    movel([0.115711, -1.231258, -2.664725, -0.816406, 1.570796, 1.686507],accel_mss,speed_ms,0,blend_radius_m)
    movel([0.117256, -1.231856, -2.664420, -0.816113, 1.570796, 1.688052],accel_mss,speed_ms,0,blend_radius_m)
    movel([0.117989, -1.233200, -2.663733, -0.815456, 1.570796, 1.688785],accel_mss,speed_ms,0,blend_radius_m)
    movel([0.117965, -1.234308, -2.663164, -0.814916, 1.570796, 1.688761],accel_mss,speed_ms,0,blend_radius_m)
    movel([0.117577, -1.235608, -2.662496, -0.814285, 1.570796, 1.688373],accel_mss,speed_ms,0,blend_radius_m)
    movel([0.116887, -1.236930, -2.661814, -0.813645, 1.570796, 1.687683],accel_mss,speed_ms,0,blend_radius_m)
    movel([0.115976, -1.238105, -2.661207, -0.813078, 1.570796, 1.686772],accel_mss,speed_ms,0,blend_radius_m)
    movel([0.115156, -1.238911, -2.660789, -0.812690, 1.570796, 1.685952],accel_mss,speed_ms,0,blend_radius_m)
    movel([0.114390, -1.239502, -2.660482, -0.812406, 1.570796, 1.685186],accel_mss,speed_ms,0,blend_radius_m)
    movel([0.113558, -1.239966, -2.660241, -0.812183, 1.570796, 1.684355],accel_mss,speed_ms,0,blend_radius_m)
    movel([0.112538, -1.240377, -2.660026, -0.811985, 1.570796, 1.683335],accel_mss,speed_ms,0,blend_radius_m)
    movel([0.111513, -1.240676, -2.659871, -0.811842, 1.570796, 1.682309],accel_mss,speed_ms,0,blend_radius_m)
    movel([0.110720, -1.240770, -2.659822, -0.811797, 1.570796, 1.681516],accel_mss,speed_ms,0,blend_radius_m)
    movel([0.110024, -1.240667, -2.659876, -0.811847, 1.570796, 1.680820],accel_mss,speed_ms,0,blend_radius_m)
    movel([0.109302, -1.240359, -2.660036, -0.811994, 1.570796, 1.680098],accel_mss,speed_ms,0,blend_radius_m)
    movel([0.108717, -1.239916, -2.660266, -0.812206, 1.570796, 1.679513],accel_mss,speed_ms,0,blend_radius_m)
    movel([0.108365, -1.239370, -2.660550, -0.812468, 1.570796, 1.679162],accel_mss,speed_ms,0,blend_radius_m)
    movel([0.108218, -1.238654, -2.660922, -0.812813, 1.570796, 1.679014],accel_mss,speed_ms,0,blend_radius_m)
    movel([0.108256, -1.237694, -2.661419, -0.813276, 1.570796, 1.679053],accel_mss,speed_ms,0,blend_radius_m)
    movel([0.108349, -1.237041, -2.661757, -0.813591, 1.570796, 1.679145],accel_mss,speed_ms,0,blend_radius_m)
    movel([0.108457, -1.236591, -2.661989, -0.813809, 1.570796, 1.679253],accel_mss,speed_ms,0,blend_radius_m)
    movel([0.108621, -1.236171, -2.662206, -0.814012, 1.570796, 1.679418],accel_mss,speed_ms,0,blend_radius_m)
    movel([0.108896, -1.235638, -2.662480, -0.814270, 1.570796, 1.679692],accel_mss,speed_ms,0,blend_radius_m)
    movel([0.109412, -1.234833, -2.662895, -0.814661, 1.570796, 1.680209],accel_mss,speed_ms,0,blend_radius_m)
    speed_ms = 0.003
    movel([0.109412, -1.220507, -2.655895, -0.835988, 1.570796, 1.680209],accel_mss,speed_ms,0,blend_radius_m)
    speed_ms = 1.000
    movel([0.109412, -1.193393, -2.641522, -0.877474, 1.570796, 1.680209],accel_mss,speed_ms,0,blend_radius_m)
    movel([0.123315, -1.189342, -2.643484, -0.879564, 1.570796, 1.694112],accel_mss,speed_ms,0,blend_radius_m)
    movel([0.123315, -1.216492, -2.657910, -0.837988, 1.570796, 1.694112],accel_mss,speed_ms,0,blend_radius_m)
    speed_ms = 0.003
    movel([0.123315, -1.227206, -2.663192, -0.821991, 1.570796, 1.694112],accel_mss,speed_ms,0,blend_radius_m)
    speed_ms = 0.007
    movel([0.123570, -1.225425, -2.664093, -0.822871, 1.570796, 1.694367],accel_mss,speed_ms,0,blend_radius_m)
    movel([0.123913, -1.223185, -2.665221, -0.823983, 1.570796, 1.694710],accel_mss,speed_ms,0,blend_radius_m)
    movel([0.124125, -1.222339, -2.665645, -0.824405, 1.570796, 1.694921],accel_mss,speed_ms,0,blend_radius_m)
    movel([0.124611, -1.222347, -2.665641, -0.824401, 1.570796, 1.695407],accel_mss,speed_ms,0,blend_radius_m)
    movel([0.124874, -1.223146, -2.665240, -0.824003, 1.570796, 1.695670],accel_mss,speed_ms,0,blend_radius_m)
    movel([0.124930, -1.224185, -2.664718, -0.823486, 1.570796, 1.695726],accel_mss,speed_ms,0,blend_radius_m)
    movel([0.124787, -1.225358, -2.664126, -0.822904, 1.570796, 1.695583],accel_mss,speed_ms,0,blend_radius_m)
    movel([0.124446, -1.226559, -2.663520, -0.822311, 1.570796, 1.695243],accel_mss,speed_ms,0,blend_radius_m)
    movel([0.124141, -1.227337, -2.663125, -0.821927, 1.570796, 1.694937],accel_mss,speed_ms,0,blend_radius_m)
    movel([0.123839, -1.227943, -2.662818, -0.821628, 1.570796, 1.694636],accel_mss,speed_ms,0,blend_radius_m)
    movel([0.123561, -1.228363, -2.662604, -0.821421, 1.570796, 1.694357],accel_mss,speed_ms,0,blend_radius_m)
    movel([0.123214, -1.228488, -2.662541, -0.821360, 1.570796, 1.694010],accel_mss,speed_ms,0,blend_radius_m)
    movel([0.123227, -1.228032, -2.662773, -0.821584, 1.570796, 1.694023],accel_mss,speed_ms,0,blend_radius_m)
    movel([0.123315, -1.227206, -2.663192, -0.821991, 1.570796, 1.694112],accel_mss,speed_ms,0,blend_radius_m)
    speed_ms = 0.003
    movel([0.123315, -1.230843, -2.664937, -0.816609, 1.570796, 1.694112],accel_mss,speed_ms,0,blend_radius_m)
    speed_ms = 0.007
    movel([0.123570, -1.229065, -2.665841, -0.817483, 1.570796, 1.694367],accel_mss,speed_ms,0,blend_radius_m)
    movel([0.123913, -1.226829, -2.666972, -0.818588, 1.570796, 1.694710],accel_mss,speed_ms,0,blend_radius_m)
    movel([0.124125, -1.225985, -2.667398, -0.819006, 1.570796, 1.694921],accel_mss,speed_ms,0,blend_radius_m)
    movel([0.124611, -1.225992, -2.667394, -0.819002, 1.570796, 1.695407],accel_mss,speed_ms,0,blend_radius_m)
    movel([0.124874, -1.226790, -2.666992, -0.818607, 1.570796, 1.695670],accel_mss,speed_ms,0,blend_radius_m)
    movel([0.124930, -1.227827, -2.666468, -0.818094, 1.570796, 1.695726],accel_mss,speed_ms,0,blend_radius_m)
    movel([0.124787, -1.228999, -2.665874, -0.817516, 1.570796, 1.695583],accel_mss,speed_ms,0,blend_radius_m)
    movel([0.124446, -1.230197, -2.665265, -0.816926, 1.570796, 1.695243],accel_mss,speed_ms,0,blend_radius_m)
    movel([0.124141, -1.230974, -2.664870, -0.816545, 1.570796, 1.694937],accel_mss,speed_ms,0,blend_radius_m)
    movel([0.123839, -1.231579, -2.664561, -0.816248, 1.570796, 1.694636],accel_mss,speed_ms,0,blend_radius_m)
    movel([0.123561, -1.231999, -2.664347, -0.816043, 1.570796, 1.694357],accel_mss,speed_ms,0,blend_radius_m)
    movel([0.123214, -1.232124, -2.664283, -0.815982, 1.570796, 1.694010],accel_mss,speed_ms,0,blend_radius_m)
    movel([0.123227, -1.231668, -2.664516, -0.816205, 1.570796, 1.694023],accel_mss,speed_ms,0,blend_radius_m)
    movel([0.123315, -1.230843, -2.664937, -0.816609, 1.570796, 1.694112],accel_mss,speed_ms,0,blend_radius_m)
    speed_ms = 0.003
    movel([0.123315, -1.216492, -2.657910, -0.837988, 1.570796, 1.694112],accel_mss,speed_ms,0,blend_radius_m)
    speed_ms = 1.000
    movel([0.123315, -1.189342, -2.643484, -0.879564, 1.570796, 1.694112],accel_mss,speed_ms,0,blend_radius_m)
    movel([0.125124, -1.188800, -2.643744, -0.879845, 1.570796, 1.695920],accel_mss,speed_ms,0,blend_radius_m)
    movel([0.125124, -1.215955, -2.658178, -0.838257, 1.570796, 1.695920],accel_mss,speed_ms,0,blend_radius_m)
    speed_ms = 0.003
    movel([0.125124, -1.226671, -2.663463, -0.822255, 1.570796, 1.695920],accel_mss,speed_ms,0,blend_radius_m)
    speed_ms = 0.007
    movel([0.125227, -1.226209, -2.663697, -0.822484, 1.570796, 1.696023],accel_mss,speed_ms,0,blend_radius_m)
    movel([0.125307, -1.225911, -2.663847, -0.822631, 1.570796, 1.696104],accel_mss,speed_ms,0,blend_radius_m)
    movel([0.125412, -1.225400, -2.664105, -0.822884, 1.570796, 1.696208],accel_mss,speed_ms,0,blend_radius_m)
    movel([0.125518, -1.224812, -2.664402, -0.823175, 1.570796, 1.696314],accel_mss,speed_ms,0,blend_radius_m)
    movel([0.125611, -1.224215, -2.664703, -0.823471, 1.570796, 1.696408],accel_mss,speed_ms,0,blend_radius_m)
    movel([0.125825, -1.222759, -2.665435, -0.824196, 1.570796, 1.696622],accel_mss,speed_ms,0,blend_radius_m)
    movel([0.126387, -1.222525, -2.665552, -0.824312, 1.570796, 1.697183],accel_mss,speed_ms,0,blend_radius_m)
    movel([0.127048, -1.222423, -2.665603, -0.824363, 1.570796, 1.697844],accel_mss,speed_ms,0,blend_radius_m)
    movel([0.127393, -1.222737, -2.665446, -0.824207, 1.570796, 1.698189],accel_mss,speed_ms,0,blend_radius_m)
    movel([0.127359, -1.223478, -2.665074, -0.823837, 1.570796, 1.698155],accel_mss,speed_ms,0,blend_radius_m)
    movel([0.126927, -1.224592, -2.664513, -0.823284, 1.570796, 1.697723],accel_mss,speed_ms,0,blend_radius_m)
    movel([0.126733, -1.224966, -2.664324, -0.823099, 1.570796, 1.697529],accel_mss,speed_ms,0,blend_radius_m)
    movel([0.126474, -1.225394, -2.664108, -0.822887, 1.570796, 1.697270],accel_mss,speed_ms,0,blend_radius_m)
    movel([0.126203, -1.225807, -2.663900, -0.822682, 1.570796, 1.696999],accel_mss,speed_ms,0,blend_radius_m)
    movel([0.125955, -1.226134, -2.663735, -0.822521, 1.570796, 1.696752],accel_mss,speed_ms,0,blend_radius_m)
    movel([0.125504, -1.226643, -2.663477, -0.822269, 1.570796, 1.696300],accel_mss,speed_ms,0,blend_radius_m)
    movel([0.125124, -1.226671, -2.663463, -0.822255, 1.570796, 1.695920],accel_mss,speed_ms,0,blend_radius_m)
    speed_ms = 0.003
    movel([0.125124, -1.230310, -2.665208, -0.816871, 1.570796, 1.695920],accel_mss,speed_ms,0,blend_radius_m)
    speed_ms = 0.007
    movel([0.125227, -1.229848, -2.665443, -0.817098, 1.570796, 1.696023],accel_mss,speed_ms,0,blend_radius_m)
    movel([0.125307, -1.229550, -2.665594, -0.817244, 1.570796, 1.696104],accel_mss,speed_ms,0,blend_radius_m)
    movel([0.125412, -1.229040, -2.665853, -0.817495, 1.570796, 1.696208],accel_mss,speed_ms,0,blend_radius_m)
    movel([0.125518, -1.228453, -2.666151, -0.817785, 1.570796, 1.696314],accel_mss,speed_ms,0,blend_radius_m)
    movel([0.125611, -1.227857, -2.666453, -0.818079, 1.570796, 1.696408],accel_mss,speed_ms,0,blend_radius_m)
    movel([0.125825, -1.226403, -2.667187, -0.818798, 1.570796, 1.696622],accel_mss,speed_ms,0,blend_radius_m)
    movel([0.126387, -1.226170, -2.667305, -0.818914, 1.570796, 1.697183],accel_mss,speed_ms,0,blend_radius_m)
    movel([0.127048, -1.226069, -2.667356, -0.818964, 1.570796, 1.697844],accel_mss,speed_ms,0,blend_radius_m)
    movel([0.127393, -1.226381, -2.667198, -0.818809, 1.570796, 1.698189],accel_mss,speed_ms,0,blend_radius_m)
    movel([0.127359, -1.227122, -2.666825, -0.818443, 1.570796, 1.698155],accel_mss,speed_ms,0,blend_radius_m)
    movel([0.126927, -1.228234, -2.666262, -0.817893, 1.570796, 1.697723],accel_mss,speed_ms,0,blend_radius_m)
    movel([0.126733, -1.228607, -2.666073, -0.817709, 1.570796, 1.697529],accel_mss,speed_ms,0,blend_radius_m)
    movel([0.126474, -1.229034, -2.665856, -0.817498, 1.570796, 1.697270],accel_mss,speed_ms,0,blend_radius_m)
    movel([0.126203, -1.229447, -2.665647, -0.817295, 1.570796, 1.696999],accel_mss,speed_ms,0,blend_radius_m)
    movel([0.125955, -1.229773, -2.665481, -0.817135, 1.570796, 1.696752],accel_mss,speed_ms,0,blend_radius_m)
    movel([0.125504, -1.230281, -2.665223, -0.816885, 1.570796, 1.696300],accel_mss,speed_ms,0,blend_radius_m)
    movel([0.125124, -1.230310, -2.665208, -0.816871, 1.570796, 1.695920],accel_mss,speed_ms,0,blend_radius_m)
    speed_ms = 0.003
    movel([0.125124, -1.215955, -2.658178, -0.838257, 1.570796, 1.695920],accel_mss,speed_ms,0,blend_radius_m)
    speed_ms = 1.000
    movel([0.125124, -1.188800, -2.643744, -0.879845, 1.570796, 1.695920],accel_mss,speed_ms,0,blend_radius_m)
    movel([0.132047, -1.189022, -2.643637, -0.879729, 1.570796, 1.702844],accel_mss,speed_ms,0,blend_radius_m)
    movel([0.132047, -1.216175, -2.658068, -0.838146, 1.570796, 1.702844],accel_mss,speed_ms,0,blend_radius_m)
    speed_ms = 0.003
    movel([0.132047, -1.226891, -2.663351, -0.822147, 1.570796, 1.702844],accel_mss,speed_ms,0,blend_radius_m)
    speed_ms = 0.007
    movel([0.132638, -1.225634, -2.663987, -0.822768, 1.570796, 1.703435],accel_mss,speed_ms,0,blend_radius_m)
    movel([0.133199, -1.224453, -2.664583, -0.823353, 1.570796, 1.703995],accel_mss,speed_ms,0,blend_radius_m)
    movel([0.133706, -1.223415, -2.665105, -0.823869, 1.570796, 1.704502],accel_mss,speed_ms,0,blend_radius_m)
    movel([0.134145, -1.222533, -2.665548, -0.824308, 1.570796, 1.704942],accel_mss,speed_ms,0,blend_radius_m)
    movel([0.134644, -1.222071, -2.665779, -0.824538, 1.570796, 1.705440],accel_mss,speed_ms,0,blend_radius_m)
    movel([0.137265, -1.221154, -2.666238, -0.824996, 1.570796, 1.708061],accel_mss,speed_ms,0,blend_radius_m)
    movel([0.139899, -1.220261, -2.666685, -0.825444, 1.570796, 1.710696],accel_mss,speed_ms,0,blend_radius_m)
    movel([0.140179, -1.220315, -2.666657, -0.825416, 1.570796, 1.710976],accel_mss,speed_ms,0,blend_radius_m)
    movel([0.139664, -1.221322, -2.666155, -0.824913, 1.570796, 1.710461],accel_mss,speed_ms,0,blend_radius_m)
    movel([0.139060, -1.222362, -2.665634, -0.824393, 1.570796, 1.709856],accel_mss,speed_ms,0,blend_radius_m)
    movel([0.138330, -1.223574, -2.665025, -0.823790, 1.570796, 1.709127],accel_mss,speed_ms,0,blend_radius_m)
    movel([0.137599, -1.224793, -2.664411, -0.823184, 1.570796, 1.708395],accel_mss,speed_ms,0,blend_radius_m)
    movel([0.136986, -1.225855, -2.663875, -0.822658, 1.570796, 1.707782],accel_mss,speed_ms,0,blend_radius_m)
    movel([0.136486, -1.226755, -2.663420, -0.822214, 1.570796, 1.707282],accel_mss,speed_ms,0,blend_radius_m)
    movel([0.136518, -1.227033, -2.663280, -0.822077, 1.570796, 1.707315],accel_mss,speed_ms,0,blend_radius_m)
    movel([0.137154, -1.226936, -2.663329, -0.822124, 1.570796, 1.707950],accel_mss,speed_ms,0,blend_radius_m)
    movel([0.138087, -1.226651, -2.663473, -0.822265, 1.570796, 1.708883],accel_mss,speed_ms,0,blend_radius_m)
    movel([0.139264, -1.226294, -2.663654, -0.822441, 1.570796, 1.710060],accel_mss,speed_ms,0,blend_radius_m)
    movel([0.139772, -1.226178, -2.663712, -0.822499, 1.570796, 1.710568],accel_mss,speed_ms,0,blend_radius_m)
    movel([0.140019, -1.226346, -2.663627, -0.822416, 1.570796, 1.710815],accel_mss,speed_ms,0,blend_radius_m)
    movel([0.138614, -1.228269, -2.662652, -0.821468, 1.570796, 1.709410],accel_mss,speed_ms,0,blend_radius_m)
    movel([0.137118, -1.230263, -2.661637, -0.820489, 1.570796, 1.707915],accel_mss,speed_ms,0,blend_radius_m)
    movel([0.135361, -1.232589, -2.660446, -0.819354, 1.570796, 1.706158],accel_mss,speed_ms,0,blend_radius_m)
    movel([0.132780, -1.235980, -2.658700, -0.817709, 1.570796, 1.703577],accel_mss,speed_ms,0,blend_radius_m)
    movel([0.131413, -1.237715, -2.657801, -0.816873, 1.570796, 1.702210],accel_mss,speed_ms,0,blend_radius_m)
    movel([0.130637, -1.238623, -2.657329, -0.816437, 1.570796, 1.701434],accel_mss,speed_ms,0,blend_radius_m)
    movel([0.131028, -1.237389, -2.657970, -0.817030, 1.570796, 1.701824],accel_mss,speed_ms,0,blend_radius_m)
    movel([0.131630, -1.236096, -2.658640, -0.817653, 1.570796, 1.702426],accel_mss,speed_ms,0,blend_radius_m)
    movel([0.132342, -1.234571, -2.659427, -0.818391, 1.570796, 1.703139],accel_mss,speed_ms,0,blend_radius_m)
    movel([0.133341, -1.232431, -2.660528, -0.819431, 1.570796, 1.704138],accel_mss,speed_ms,0,blend_radius_m)
    movel([0.133828, -1.231324, -2.661095, -0.819971, 1.570796, 1.704624],accel_mss,speed_ms,0,blend_radius_m)
    movel([0.134081, -1.230655, -2.661436, -0.820297, 1.570796, 1.704877],accel_mss,speed_ms,0,blend_radius_m)
    movel([0.133888, -1.230404, -2.661565, -0.820420, 1.570796, 1.704685],accel_mss,speed_ms,0,blend_radius_m)
    movel([0.133543, -1.230462, -2.661535, -0.820392, 1.570796, 1.704340],accel_mss,speed_ms,0,blend_radius_m)
    movel([0.132977, -1.230620, -2.661454, -0.820314, 1.570796, 1.703773],accel_mss,speed_ms,0,blend_radius_m)
    movel([0.131976, -1.230948, -2.661287, -0.820154, 1.570796, 1.702773],accel_mss,speed_ms,0,blend_radius_m)
    movel([0.131026, -1.231259, -2.661128, -0.820002, 1.570796, 1.701823],accel_mss,speed_ms,0,blend_radius_m)
    movel([0.130463, -1.231420, -2.661045, -0.819923, 1.570796, 1.701259],accel_mss,speed_ms,0,blend_radius_m)
    movel([0.130111, -1.231489, -2.661010, -0.819890, 1.570796, 1.700907],accel_mss,speed_ms,0,blend_radius_m)
    movel([0.130157, -1.230942, -2.661290, -0.820157, 1.570796, 1.700954],accel_mss,speed_ms,0,blend_radius_m)
    movel([0.130350, -1.230484, -2.661524, -0.820381, 1.570796, 1.701146],accel_mss,speed_ms,0,blend_radius_m)
    movel([0.130587, -1.229971, -2.661786, -0.820632, 1.570796, 1.701384],accel_mss,speed_ms,0,blend_radius_m)
    movel([0.130923, -1.229270, -2.662143, -0.820976, 1.570796, 1.701719],accel_mss,speed_ms,0,blend_radius_m)
    movel([0.131451, -1.228156, -2.662710, -0.821523, 1.570796, 1.702247],accel_mss,speed_ms,0,blend_radius_m)
    movel([0.132047, -1.226891, -2.663351, -0.822147, 1.570796, 1.702844],accel_mss,speed_ms,0,blend_radius_m)
    speed_ms = 0.003
    movel([0.132047, -1.230529, -2.665097, -0.816763, 1.570796, 1.702844],accel_mss,speed_ms,0,blend_radius_m)
    speed_ms = 0.007
    movel([0.132638, -1.229274, -2.665735, -0.817380, 1.570796, 1.703435],accel_mss,speed_ms,0,blend_radius_m)
    movel([0.133199, -1.228095, -2.666332, -0.817962, 1.570796, 1.703995],accel_mss,speed_ms,0,blend_radius_m)
    movel([0.133706, -1.227059, -2.666856, -0.818474, 1.570796, 1.704502],accel_mss,speed_ms,0,blend_radius_m)
    movel([0.134145, -1.226178, -2.667301, -0.818910, 1.570796, 1.704942],accel_mss,speed_ms,0,blend_radius_m)
    movel([0.134644, -1.225717, -2.667533, -0.819139, 1.570796, 1.705440],accel_mss,speed_ms,0,blend_radius_m)
    movel([0.137265, -1.224801, -2.667994, -0.819594, 1.570796, 1.708061],accel_mss,speed_ms,0,blend_radius_m)
    movel([0.139899, -1.223910, -2.668441, -0.820038, 1.570796, 1.710696],accel_mss,speed_ms,0,blend_radius_m)
    movel([0.140179, -1.223964, -2.668414, -0.820011, 1.570796, 1.710976],accel_mss,speed_ms,0,blend_radius_m)
    movel([0.139664, -1.224969, -2.667909, -0.819511, 1.570796, 1.710461],accel_mss,speed_ms,0,blend_radius_m)
    movel([0.139060, -1.226007, -2.667387, -0.818995, 1.570796, 1.709856],accel_mss,speed_ms,0,blend_radius_m)
    movel([0.138330, -1.227218, -2.666776, -0.818395, 1.570796, 1.709127],accel_mss,speed_ms,0,blend_radius_m)
    movel([0.137599, -1.228435, -2.666160, -0.817794, 1.570796, 1.708395],accel_mss,speed_ms,0,blend_radius_m)
    movel([0.136986, -1.229495, -2.665622, -0.817271, 1.570796, 1.707782],accel_mss,speed_ms,0,blend_radius_m)
    movel([0.136486, -1.230393, -2.665166, -0.816830, 1.570796, 1.707282],accel_mss,speed_ms,0,blend_radius_m)
    movel([0.136518, -1.230670, -2.665025, -0.816694, 1.570796, 1.707315],accel_mss,speed_ms,0,blend_radius_m)
    movel([0.137154, -1.230574, -2.665074, -0.816741, 1.570796, 1.707950],accel_mss,speed_ms,0,blend_radius_m)
    movel([0.138087, -1.230290, -2.665218, -0.816881, 1.570796, 1.708883],accel_mss,speed_ms,0,blend_radius_m)
    movel([0.139264, -1.229933, -2.665400, -0.817056, 1.570796, 1.710060],accel_mss,speed_ms,0,blend_radius_m)
    movel([0.139772, -1.229817, -2.665459, -0.817113, 1.570796, 1.710568],accel_mss,speed_ms,0,blend_radius_m)
    movel([0.140019, -1.229985, -2.665374, -0.817031, 1.570796, 1.710815],accel_mss,speed_ms,0,blend_radius_m)
    movel([0.138614, -1.231905, -2.664395, -0.816089, 1.570796, 1.709410],accel_mss,speed_ms,0,blend_radius_m)
    movel([0.137118, -1.233896, -2.663376, -0.815117, 1.570796, 1.707915],accel_mss,speed_ms,0,blend_radius_m)
    movel([0.135361, -1.236217, -2.662182, -0.813990, 1.570796, 1.706158],accel_mss,speed_ms,0,blend_radius_m)
    movel([0.132780, -1.239602, -2.660430, -0.812357, 1.570796, 1.703577],accel_mss,speed_ms,0,blend_radius_m)
    movel([0.131413, -1.241335, -2.659528, -0.811527, 1.570796, 1.702210],accel_mss,speed_ms,0,blend_radius_m)
    movel([0.130637, -1.242241, -2.659054, -0.811094, 1.570796, 1.701434],accel_mss,speed_ms,0,blend_radius_m)
    movel([0.131028, -1.241009, -2.659697, -0.811683, 1.570796, 1.701824],accel_mss,speed_ms,0,blend_radius_m)
    movel([0.131630, -1.239718, -2.660369, -0.812302, 1.570796, 1.702426],accel_mss,speed_ms,0,blend_radius_m)
    movel([0.132342, -1.238196, -2.661159, -0.813034, 1.570796, 1.703139],accel_mss,speed_ms,0,blend_radius_m)
    movel([0.133341, -1.236060, -2.662263, -0.814066, 1.570796, 1.704138],accel_mss,speed_ms,0,blend_radius_m)
    movel([0.133828, -1.234954, -2.662832, -0.814602, 1.570796, 1.704624],accel_mss,speed_ms,0,blend_radius_m)
    movel([0.134081, -1.234287, -2.663175, -0.814927, 1.570796, 1.704877],accel_mss,speed_ms,0,blend_radius_m)
    movel([0.133888, -1.234036, -2.663304, -0.815049, 1.570796, 1.704685],accel_mss,speed_ms,0,blend_radius_m)
    movel([0.133543, -1.234094, -2.663274, -0.815021, 1.570796, 1.704340],accel_mss,speed_ms,0,blend_radius_m)
    movel([0.132977, -1.234252, -2.663193, -0.814944, 1.570796, 1.703773],accel_mss,speed_ms,0,blend_radius_m)
    movel([0.131976, -1.234579, -2.663025, -0.814785, 1.570796, 1.702773],accel_mss,speed_ms,0,blend_radius_m)
    movel([0.131026, -1.234890, -2.662866, -0.814634, 1.570796, 1.701823],accel_mss,speed_ms,0,blend_radius_m)
    movel([0.130463, -1.235050, -2.662783, -0.814556, 1.570796, 1.701259],accel_mss,speed_ms,0,blend_radius_m)
    movel([0.130111, -1.235119, -2.662747, -0.814522, 1.570796, 1.700907],accel_mss,speed_ms,0,blend_radius_m)
    movel([0.130157, -1.234573, -2.663028, -0.814787, 1.570796, 1.700954],accel_mss,speed_ms,0,blend_radius_m)
    movel([0.130350, -1.234116, -2.663263, -0.815010, 1.570796, 1.701146],accel_mss,speed_ms,0,blend_radius_m)
    movel([0.130587, -1.233603, -2.663526, -0.815260, 1.570796, 1.701384],accel_mss,speed_ms,0,blend_radius_m)
    movel([0.130923, -1.232904, -2.663884, -0.815601, 1.570796, 1.701719],accel_mss,speed_ms,0,blend_radius_m)
    movel([0.131451, -1.231792, -2.664453, -0.816144, 1.570796, 1.702247],accel_mss,speed_ms,0,blend_radius_m)
    movel([0.132047, -1.230529, -2.665097, -0.816763, 1.570796, 1.702844],accel_mss,speed_ms,0,blend_radius_m)
    speed_ms = 0.003
    movel([0.132047, -1.216175, -2.658068, -0.838146, 1.570796, 1.702844],accel_mss,speed_ms,0,blend_radius_m)
    speed_ms = 1.000
    movel([0.132047, -1.189022, -2.643637, -0.879729, 1.570796, 1.702844],accel_mss,speed_ms,0,blend_radius_m)
    movel([0.137167, -1.179616, -2.648120, -0.884653, 1.570796, 1.707964],accel_mss,speed_ms,0,blend_radius_m)
    movel([0.137167, -1.206848, -2.662674, -0.842866, 1.570796, 1.707964],accel_mss,speed_ms,0,blend_radius_m)
    speed_ms = 0.003
    movel([0.137167, -1.217605, -2.668006, -0.826778, 1.570796, 1.707964],accel_mss,speed_ms,0,blend_radius_m)
    speed_ms = 0.007
    movel([0.132044, -1.218458, -2.667582, -0.826349, 1.570796, 1.702840],accel_mss,speed_ms,0,blend_radius_m)
    movel([0.128297, -1.219090, -2.667268, -0.826031, 1.570796, 1.699093],accel_mss,speed_ms,0,blend_radius_m)
    movel([0.127537, -1.219189, -2.667219, -0.825981, 1.570796, 1.698333],accel_mss,speed_ms,0,blend_radius_m)
    movel([0.127058, -1.219267, -2.667180, -0.825942, 1.570796, 1.697854],accel_mss,speed_ms,0,blend_radius_m)
    movel([0.126617, -1.219381, -2.667123, -0.825885, 1.570796, 1.697414],accel_mss,speed_ms,0,blend_radius_m)
    movel([0.126265, -1.219434, -2.667097, -0.825858, 1.570796, 1.697062],accel_mss,speed_ms,0,blend_radius_m)
    movel([0.126070, -1.219309, -2.667159, -0.825921, 1.570796, 1.696867],accel_mss,speed_ms,0,blend_radius_m)
    movel([0.126087, -1.219038, -2.667294, -0.826057, 1.570796, 1.696884],accel_mss,speed_ms,0,blend_radius_m)
    movel([0.126310, -1.218696, -2.667464, -0.826229, 1.570796, 1.697106],accel_mss,speed_ms,0,blend_radius_m)
    movel([0.126663, -1.218384, -2.667619, -0.826386, 1.570796, 1.697459],accel_mss,speed_ms,0,blend_radius_m)
    movel([0.127031, -1.218177, -2.667722, -0.826490, 1.570796, 1.697827],accel_mss,speed_ms,0,blend_radius_m)
    movel([0.127409, -1.217915, -2.667852, -0.826622, 1.570796, 1.698205],accel_mss,speed_ms,0,blend_radius_m)
    movel([0.127262, -1.217624, -2.667996, -0.826769, 1.570796, 1.698059],accel_mss,speed_ms,0,blend_radius_m)
    movel([0.127149, -1.217345, -2.668135, -0.826910, 1.570796, 1.697945],accel_mss,speed_ms,0,blend_radius_m)
    movel([0.127428, -1.216453, -2.668576, -0.827360, 1.570796, 1.698224],accel_mss,speed_ms,0,blend_radius_m)
    movel([0.127659, -1.215739, -2.668929, -0.827721, 1.570796, 1.698456],accel_mss,speed_ms,0,blend_radius_m)
    movel([0.127920, -1.214942, -2.669322, -0.828125, 1.570796, 1.698716],accel_mss,speed_ms,0,blend_radius_m)
    movel([0.128552, -1.213077, -2.670239, -0.829072, 1.570796, 1.699349],accel_mss,speed_ms,0,blend_radius_m)
    movel([0.129233, -1.211228, -2.671145, -0.830016, 1.570796, 1.700029],accel_mss,speed_ms,0,blend_radius_m)
    movel([0.129919, -1.209504, -2.671986, -0.830899, 1.570796, 1.700715],accel_mss,speed_ms,0,blend_radius_m)
    movel([0.130573, -1.208010, -2.672712, -0.831667, 1.570796, 1.701370],accel_mss,speed_ms,0,blend_radius_m)
    movel([0.131186, -1.206763, -2.673316, -0.832310, 1.570796, 1.701982],accel_mss,speed_ms,0,blend_radius_m)
    movel([0.131992, -1.205264, -2.674040, -0.833085, 1.570796, 1.702789],accel_mss,speed_ms,0,blend_radius_m)
    movel([0.132796, -1.203858, -2.674717, -0.833814, 1.570796, 1.703592],accel_mss,speed_ms,0,blend_radius_m)
    movel([0.133240, -1.203225, -2.675021, -0.834143, 1.570796, 1.704036],accel_mss,speed_ms,0,blend_radius_m)
    movel([0.133419, -1.202909, -2.675172, -0.834307, 1.570796, 1.704215],accel_mss,speed_ms,0,blend_radius_m)
    movel([0.133141, -1.202717, -2.675264, -0.834408, 1.570796, 1.703937],accel_mss,speed_ms,0,blend_radius_m)
    movel([0.132854, -1.202460, -2.675388, -0.834542, 1.570796, 1.703650],accel_mss,speed_ms,0,blend_radius_m)
    movel([0.132762, -1.202006, -2.675605, -0.834778, 1.570796, 1.703558],accel_mss,speed_ms,0,blend_radius_m)
    movel([0.132845, -1.201523, -2.675836, -0.835030, 1.570796, 1.703642],accel_mss,speed_ms,0,blend_radius_m)
    movel([0.133091, -1.201115, -2.676031, -0.835243, 1.570796, 1.703887],accel_mss,speed_ms,0,blend_radius_m)
    movel([0.133535, -1.200749, -2.676206, -0.835435, 1.570796, 1.704331],accel_mss,speed_ms,0,blend_radius_m)
    movel([0.134241, -1.200375, -2.676384, -0.835630, 1.570796, 1.705037],accel_mss,speed_ms,0,blend_radius_m)
    movel([0.134764, -1.200111, -2.676510, -0.835768, 1.570796, 1.705560],accel_mss,speed_ms,0,blend_radius_m)
    movel([0.135062, -1.199709, -2.676701, -0.835979, 1.570796, 1.705858],accel_mss,speed_ms,0,blend_radius_m)
    movel([0.134891, -1.199556, -2.676774, -0.836059, 1.570796, 1.705688],accel_mss,speed_ms,0,blend_radius_m)
    movel([0.134732, -1.199225, -2.676931, -0.836232, 1.570796, 1.705528],accel_mss,speed_ms,0,blend_radius_m)
    movel([0.135045, -1.198659, -2.677200, -0.836530, 1.570796, 1.705842],accel_mss,speed_ms,0,blend_radius_m)
    movel([0.135260, -1.198332, -2.677355, -0.836702, 1.570796, 1.706056],accel_mss,speed_ms,0,blend_radius_m)
    movel([0.135106, -1.198121, -2.677455, -0.836812, 1.570796, 1.705902],accel_mss,speed_ms,0,blend_radius_m)
    movel([0.134979, -1.197887, -2.677566, -0.836935, 1.570796, 1.705775],accel_mss,speed_ms,0,blend_radius_m)
    movel([0.135022, -1.197549, -2.677726, -0.837113, 1.570796, 1.705819],accel_mss,speed_ms,0,blend_radius_m)
    movel([0.135228, -1.197162, -2.677910, -0.837317, 1.570796, 1.706025],accel_mss,speed_ms,0,blend_radius_m)
    movel([0.135563, -1.196794, -2.678084, -0.837511, 1.570796, 1.706360],accel_mss,speed_ms,0,blend_radius_m)
    movel([0.136122, -1.196424, -2.678259, -0.837706, 1.570796, 1.706918],accel_mss,speed_ms,0,blend_radius_m)
    movel([0.136520, -1.196210, -2.678360, -0.837819, 1.570796, 1.707316],accel_mss,speed_ms,0,blend_radius_m)
    movel([0.136917, -1.196020, -2.678449, -0.837920, 1.570796, 1.707713],accel_mss,speed_ms,0,blend_radius_m)
    movel([0.137667, -1.195725, -2.678589, -0.838075, 1.570796, 1.708464],accel_mss,speed_ms,0,blend_radius_m)
    movel([0.138053, -1.195693, -2.678604, -0.838092, 1.570796, 1.708850],accel_mss,speed_ms,0,blend_radius_m)
    movel([0.138221, -1.195886, -2.678512, -0.837990, 1.570796, 1.709017],accel_mss,speed_ms,0,blend_radius_m)
    movel([0.138216, -1.196354, -2.678292, -0.837743, 1.570796, 1.709012],accel_mss,speed_ms,0,blend_radius_m)
    movel([0.138152, -1.196689, -2.678133, -0.837566, 1.570796, 1.708948],accel_mss,speed_ms,0,blend_radius_m)
    movel([0.137928, -1.197009, -2.677982, -0.837398, 1.570796, 1.708725],accel_mss,speed_ms,0,blend_radius_m)
    movel([0.137210, -1.197431, -2.677782, -0.837175, 1.570796, 1.708006],accel_mss,speed_ms,0,blend_radius_m)
    movel([0.137030, -1.197760, -2.677627, -0.837002, 1.570796, 1.707826],accel_mss,speed_ms,0,blend_radius_m)
    movel([0.137325, -1.197719, -2.677646, -0.837024, 1.570796, 1.708122],accel_mss,speed_ms,0,blend_radius_m)
    movel([0.137916, -1.197664, -2.677672, -0.837053, 1.570796, 1.708712],accel_mss,speed_ms,0,blend_radius_m)
    movel([0.138103, -1.197922, -2.677550, -0.836917, 1.570796, 1.708899],accel_mss,speed_ms,0,blend_radius_m)
    movel([0.137849, -1.198333, -2.677355, -0.836701, 1.570796, 1.708645],accel_mss,speed_ms,0,blend_radius_m)
    movel([0.137229, -1.198709, -2.677176, -0.836503, 1.570796, 1.708025],accel_mss,speed_ms,0,blend_radius_m)
    movel([0.136800, -1.198942, -2.677066, -0.836381, 1.570796, 1.707596],accel_mss,speed_ms,0,blend_radius_m)
    movel([0.137077, -1.199164, -2.676960, -0.836265, 1.570796, 1.707873],accel_mss,speed_ms,0,blend_radius_m)
    movel([0.137743, -1.198969, -2.677053, -0.836367, 1.570796, 1.708539],accel_mss,speed_ms,0,blend_radius_m)
    movel([0.139062, -1.198526, -2.677263, -0.836600, 1.570796, 1.709859],accel_mss,speed_ms,0,blend_radius_m)
    movel([0.140035, -1.198197, -2.677419, -0.836773, 1.570796, 1.710832],accel_mss,speed_ms,0,blend_radius_m)
    movel([0.140925, -1.197898, -2.677561, -0.836930, 1.570796, 1.711721],accel_mss,speed_ms,0,blend_radius_m)
    movel([0.141673, -1.197645, -2.677681, -0.837063, 1.570796, 1.712470],accel_mss,speed_ms,0,blend_radius_m)
    movel([0.142196, -1.197458, -2.677770, -0.837161, 1.570796, 1.712992],accel_mss,speed_ms,0,blend_radius_m)
    movel([0.142396, -1.196953, -2.678008, -0.837427, 1.570796, 1.713192],accel_mss,speed_ms,0,blend_radius_m)
    movel([0.142482, -1.196504, -2.678221, -0.837664, 1.570796, 1.713278],accel_mss,speed_ms,0,blend_radius_m)
    movel([0.142693, -1.196175, -2.678376, -0.837838, 1.570796, 1.713489],accel_mss,speed_ms,0,blend_radius_m)
    movel([0.143073, -1.195909, -2.678502, -0.837978, 1.570796, 1.713870],accel_mss,speed_ms,0,blend_radius_m)
    movel([0.143726, -1.195644, -2.678627, -0.838118, 1.570796, 1.714522],accel_mss,speed_ms,0,blend_radius_m)
    movel([0.144613, -1.195393, -2.678745, -0.838251, 1.570796, 1.715409],accel_mss,speed_ms,0,blend_radius_m)
    movel([0.146289, -1.195058, -2.678903, -0.838428, 1.570796, 1.717085],accel_mss,speed_ms,0,blend_radius_m)
    movel([0.148054, -1.194752, -2.679047, -0.838590, 1.570796, 1.718850],accel_mss,speed_ms,0,blend_radius_m)
    movel([0.149467, -1.194567, -2.679134, -0.838688, 1.570796, 1.720263],accel_mss,speed_ms,0,blend_radius_m)
    movel([0.150215, -1.194563, -2.679136, -0.838690, 1.570796, 1.721012],accel_mss,speed_ms,0,blend_radius_m)
    movel([0.150569, -1.194781, -2.679033, -0.838575, 1.570796, 1.721365],accel_mss,speed_ms,0,blend_radius_m)
    movel([0.150549, -1.195195, -2.678838, -0.838356, 1.570796, 1.721345],accel_mss,speed_ms,0,blend_radius_m)
    movel([0.150172, -1.195794, -2.678556, -0.838039, 1.570796, 1.720969],accel_mss,speed_ms,0,blend_radius_m)
    movel([0.149950, -1.196125, -2.678400, -0.837864, 1.570796, 1.720746],accel_mss,speed_ms,0,blend_radius_m)
    movel([0.150186, -1.196198, -2.678365, -0.837826, 1.570796, 1.720983],accel_mss,speed_ms,0,blend_radius_m)
    movel([0.151955, -1.196137, -2.678394, -0.837858, 1.570796, 1.722751],accel_mss,speed_ms,0,blend_radius_m)
    movel([0.153640, -1.196066, -2.678428, -0.837895, 1.570796, 1.724436],accel_mss,speed_ms,0,blend_radius_m)
    movel([0.154196, -1.195996, -2.678461, -0.837932, 1.570796, 1.724992],accel_mss,speed_ms,0,blend_radius_m)
    movel([0.154590, -1.195888, -2.678512, -0.837989, 1.570796, 1.725386],accel_mss,speed_ms,0,blend_radius_m)
    movel([0.154444, -1.195516, -2.678687, -0.838186, 1.570796, 1.725241],accel_mss,speed_ms,0,blend_radius_m)
    movel([0.154519, -1.195136, -2.678866, -0.838387, 1.570796, 1.725315],accel_mss,speed_ms,0,blend_radius_m)
    movel([0.154747, -1.194759, -2.679044, -0.838586, 1.570796, 1.725543],accel_mss,speed_ms,0,blend_radius_m)
    movel([0.155058, -1.194522, -2.679155, -0.838712, 1.570796, 1.725854],accel_mss,speed_ms,0,blend_radius_m)
    movel([0.155384, -1.194381, -2.679221, -0.838787, 1.570796, 1.726181],accel_mss,speed_ms,0,blend_radius_m)
    movel([0.155303, -1.193888, -2.679453, -0.839048, 1.570796, 1.726099],accel_mss,speed_ms,0,blend_radius_m)
    movel([0.155399, -1.193519, -2.679626, -0.839244, 1.570796, 1.726195],accel_mss,speed_ms,0,blend_radius_m)
    movel([0.155618, -1.193133, -2.679807, -0.839449, 1.570796, 1.726414],accel_mss,speed_ms,0,blend_radius_m)
    movel([0.155910, -1.192832, -2.679948, -0.839608, 1.570796, 1.726707],accel_mss,speed_ms,0,blend_radius_m)
    movel([0.156578, -1.192540, -2.680085, -0.839764, 1.570796, 1.727375],accel_mss,speed_ms,0,blend_radius_m)
    movel([0.157432, -1.192592, -2.680061, -0.839736, 1.570796, 1.728228],accel_mss,speed_ms,0,blend_radius_m)
    movel([0.158123, -1.192890, -2.679921, -0.839578, 1.570796, 1.728920],accel_mss,speed_ms,0,blend_radius_m)
    movel([0.158279, -1.193368, -2.679697, -0.839324, 1.570796, 1.729075],accel_mss,speed_ms,0,blend_radius_m)
    movel([0.158145, -1.193714, -2.679535, -0.839141, 1.570796, 1.728941],accel_mss,speed_ms,0,blend_radius_m)
    movel([0.157855, -1.194117, -2.679346, -0.838927, 1.570796, 1.728652],accel_mss,speed_ms,0,blend_radius_m)
    movel([0.157522, -1.194436, -2.679196, -0.838758, 1.570796, 1.728318],accel_mss,speed_ms,0,blend_radius_m)
    movel([0.157209, -1.194563, -2.679136, -0.838690, 1.570796, 1.728005],accel_mss,speed_ms,0,blend_radius_m)
    movel([0.157324, -1.194849, -2.679001, -0.838539, 1.570796, 1.728120],accel_mss,speed_ms,0,blend_radius_m)
    movel([0.157482, -1.195055, -2.678904, -0.838430, 1.570796, 1.728278],accel_mss,speed_ms,0,blend_radius_m)
    movel([0.157265, -1.195546, -2.678673, -0.838170, 1.570796, 1.728062],accel_mss,speed_ms,0,blend_radius_m)
    movel([0.156939, -1.195859, -2.678525, -0.838005, 1.570796, 1.727736],accel_mss,speed_ms,0,blend_radius_m)
    movel([0.156605, -1.196081, -2.678421, -0.837887, 1.570796, 1.727401],accel_mss,speed_ms,0,blend_radius_m)
    movel([0.156890, -1.196434, -2.678254, -0.837701, 1.570796, 1.727686],accel_mss,speed_ms,0,blend_radius_m)
    movel([0.157140, -1.196517, -2.678215, -0.837657, 1.570796, 1.727937],accel_mss,speed_ms,0,blend_radius_m)
    movel([0.157374, -1.196615, -2.678168, -0.837606, 1.570796, 1.728170],accel_mss,speed_ms,0,blend_radius_m)
    movel([0.157666, -1.196781, -2.678090, -0.837518, 1.570796, 1.728462],accel_mss,speed_ms,0,blend_radius_m)
    movel([0.157753, -1.197298, -2.677845, -0.837245, 1.570796, 1.728550],accel_mss,speed_ms,0,blend_radius_m)
    movel([0.157631, -1.197663, -2.677673, -0.837053, 1.570796, 1.728427],accel_mss,speed_ms,0,blend_radius_m)
    movel([0.157410, -1.198044, -2.677492, -0.836853, 1.570796, 1.728206],accel_mss,speed_ms,0,blend_radius_m)
    movel([0.157110, -1.198413, -2.677317, -0.836659, 1.570796, 1.727906],accel_mss,speed_ms,0,blend_radius_m)
    movel([0.156493, -1.198750, -2.677157, -0.836482, 1.570796, 1.727289],accel_mss,speed_ms,0,blend_radius_m)
    movel([0.155987, -1.198807, -2.677130, -0.836452, 1.570796, 1.726784],accel_mss,speed_ms,0,blend_radius_m)
    movel([0.155517, -1.198841, -2.677114, -0.836434, 1.570796, 1.726313],accel_mss,speed_ms,0,blend_radius_m)
    movel([0.156081, -1.199170, -2.676958, -0.836262, 1.570796, 1.726877],accel_mss,speed_ms,0,blend_radius_m)
    movel([0.156250, -1.199699, -2.676706, -0.835984, 1.570796, 1.727047],accel_mss,speed_ms,0,blend_radius_m)
    movel([0.156200, -1.200748, -2.676206, -0.835435, 1.570796, 1.726996],accel_mss,speed_ms,0,blend_radius_m)
    movel([0.155879, -1.202862, -2.675195, -0.834332, 1.570796, 1.726675],accel_mss,speed_ms,0,blend_radius_m)
    movel([0.155597, -1.204465, -2.674425, -0.833499, 1.570796, 1.726393],accel_mss,speed_ms,0,blend_radius_m)
    movel([0.155343, -1.205675, -2.673842, -0.832872, 1.570796, 1.726140],accel_mss,speed_ms,0,blend_radius_m)
    movel([0.155059, -1.206793, -2.673302, -0.832294, 1.570796, 1.725856],accel_mss,speed_ms,0,blend_radius_m)
    movel([0.154680, -1.208072, -2.672682, -0.831635, 1.570796, 1.725476],accel_mss,speed_ms,0,blend_radius_m)
    movel([0.153984, -1.210241, -2.671627, -0.830521, 1.570796, 1.724781],accel_mss,speed_ms,0,blend_radius_m)
    movel([0.153418, -1.211864, -2.670834, -0.829691, 1.570796, 1.724214],accel_mss,speed_ms,0,blend_radius_m)
    movel([0.152953, -1.213071, -2.670242, -0.829075, 1.570796, 1.723749],accel_mss,speed_ms,0,blend_radius_m)
    movel([0.152673, -1.213520, -2.670022, -0.828847, 1.570796, 1.723469],accel_mss,speed_ms,0,blend_radius_m)
    movel([0.152497, -1.213824, -2.669873, -0.828692, 1.570796, 1.723293],accel_mss,speed_ms,0,blend_radius_m)
    movel([0.152728, -1.214072, -2.669751, -0.828566, 1.570796, 1.723524],accel_mss,speed_ms,0,blend_radius_m)
    movel([0.152948, -1.214300, -2.669638, -0.828450, 1.570796, 1.723744],accel_mss,speed_ms,0,blend_radius_m)
    movel([0.152699, -1.214893, -2.669347, -0.828150, 1.570796, 1.723495],accel_mss,speed_ms,0,blend_radius_m)
    movel([0.151831, -1.215185, -2.669203, -0.828001, 1.570796, 1.722627],accel_mss,speed_ms,0,blend_radius_m)
    movel([0.150034, -1.215529, -2.669033, -0.827827, 1.570796, 1.720831],accel_mss,speed_ms,0,blend_radius_m)
    movel([0.144850, -1.216355, -2.668625, -0.827409, 1.570796, 1.715647],accel_mss,speed_ms,0,blend_radius_m)
    movel([0.137167, -1.217605, -2.668006, -0.826778, 1.570796, 1.707964],accel_mss,speed_ms,0,blend_radius_m)
    speed_ms = 0.003
    movel([0.137167, -1.221258, -2.669767, -0.821364, 1.570796, 1.707964],accel_mss,speed_ms,0,blend_radius_m)
    speed_ms = 0.007
    movel([0.132044, -1.222110, -2.669342, -0.820937, 1.570796, 1.702840],accel_mss,speed_ms,0,blend_radius_m)
    movel([0.128297, -1.222740, -2.669027, -0.820622, 1.570796, 1.699093],accel_mss,speed_ms,0,blend_radius_m)
    movel([0.127537, -1.222839, -2.668977, -0.820573, 1.570796, 1.698333],accel_mss,speed_ms,0,blend_radius_m)
    movel([0.127058, -1.222918, -2.668938, -0.820533, 1.570796, 1.697854],accel_mss,speed_ms,0,blend_radius_m)
    movel([0.126617, -1.223031, -2.668881, -0.820477, 1.570796, 1.697414],accel_mss,speed_ms,0,blend_radius_m)
    movel([0.126265, -1.223084, -2.668855, -0.820450, 1.570796, 1.697062],accel_mss,speed_ms,0,blend_radius_m)
    movel([0.126070, -1.222959, -2.668917, -0.820513, 1.570796, 1.696867],accel_mss,speed_ms,0,blend_radius_m)
    movel([0.126087, -1.222689, -2.669053, -0.820648, 1.570796, 1.696884],accel_mss,speed_ms,0,blend_radius_m)
    movel([0.126310, -1.222347, -2.669224, -0.820819, 1.570796, 1.697106],accel_mss,speed_ms,0,blend_radius_m)
    movel([0.126663, -1.222036, -2.669379, -0.820974, 1.570796, 1.697459],accel_mss,speed_ms,0,blend_radius_m)
    movel([0.127031, -1.221829, -2.669482, -0.821078, 1.570796, 1.697827],accel_mss,speed_ms,0,blend_radius_m)
    movel([0.127409, -1.221568, -2.669612, -0.821209, 1.570796, 1.698205],accel_mss,speed_ms,0,blend_radius_m)
    movel([0.127262, -1.221277, -2.669757, -0.821355, 1.570796, 1.698059],accel_mss,speed_ms,0,blend_radius_m)
    movel([0.127149, -1.220998, -2.669896, -0.821495, 1.570796, 1.697945],accel_mss,speed_ms,0,blend_radius_m)
    movel([0.127428, -1.220108, -2.670339, -0.821942, 1.570796, 1.698224],accel_mss,speed_ms,0,blend_radius_m)
    movel([0.127659, -1.219395, -2.670693, -0.822301, 1.570796, 1.698456],accel_mss,speed_ms,0,blend_radius_m)
    movel([0.127920, -1.218599, -2.671088, -0.822702, 1.570796, 1.698716],accel_mss,speed_ms,0,blend_radius_m)
    movel([0.128552, -1.216737, -2.672008, -0.823643, 1.570796, 1.699349],accel_mss,speed_ms,0,blend_radius_m)
    movel([0.129233, -1.214891, -2.672917, -0.824581, 1.570796, 1.700029],accel_mss,speed_ms,0,blend_radius_m)
    movel([0.129919, -1.213169, -2.673761, -0.825459, 1.570796, 1.700715],accel_mss,speed_ms,0,blend_radius_m)
    movel([0.130573, -1.211677, -2.674490, -0.826222, 1.570796, 1.701370],accel_mss,speed_ms,0,blend_radius_m)
    movel([0.131186, -1.210432, -2.675096, -0.826861, 1.570796, 1.701982],accel_mss,speed_ms,0,blend_radius_m)
    movel([0.131992, -1.208935, -2.675823, -0.827631, 1.570796, 1.702789],accel_mss,speed_ms,0,blend_radius_m)
    movel([0.132796, -1.207531, -2.676502, -0.828356, 1.570796, 1.703592],accel_mss,speed_ms,0,blend_radius_m)
    movel([0.133240, -1.206899, -2.676807, -0.828683, 1.570796, 1.704036],accel_mss,speed_ms,0,blend_radius_m)
    movel([0.133419, -1.206584, -2.676959, -0.828846, 1.570796, 1.704215],accel_mss,speed_ms,0,blend_radius_m)
    movel([0.133141, -1.206392, -2.677051, -0.828946, 1.570796, 1.703937],accel_mss,speed_ms,0,blend_radius_m)
    movel([0.132854, -1.206135, -2.677175, -0.829079, 1.570796, 1.703650],accel_mss,speed_ms,0,blend_radius_m)
    movel([0.132762, -1.205682, -2.677393, -0.829314, 1.570796, 1.703558],accel_mss,speed_ms,0,blend_radius_m)
    movel([0.132845, -1.205200, -2.677625, -0.829565, 1.570796, 1.703642],accel_mss,speed_ms,0,blend_radius_m)
    movel([0.133091, -1.204793, -2.677820, -0.829776, 1.570796, 1.703887],accel_mss,speed_ms,0,blend_radius_m)
    movel([0.133535, -1.204427, -2.677996, -0.829967, 1.570796, 1.704331],accel_mss,speed_ms,0,blend_radius_m)
    movel([0.134241, -1.204053, -2.678175, -0.830161, 1.570796, 1.705037],accel_mss,speed_ms,0,blend_radius_m)
    movel([0.134764, -1.203790, -2.678301, -0.830298, 1.570796, 1.705560],accel_mss,speed_ms,0,blend_radius_m)
    movel([0.135062, -1.203388, -2.678493, -0.830508, 1.570796, 1.705858],accel_mss,speed_ms,0,blend_radius_m)
    movel([0.134891, -1.203236, -2.678566, -0.830587, 1.570796, 1.705688],accel_mss,speed_ms,0,blend_radius_m)
    movel([0.134732, -1.202905, -2.678724, -0.830760, 1.570796, 1.705528],accel_mss,speed_ms,0,blend_radius_m)
    movel([0.135045, -1.202340, -2.678994, -0.831055, 1.570796, 1.705842],accel_mss,speed_ms,0,blend_radius_m)
    movel([0.135260, -1.202013, -2.679150, -0.831226, 1.570796, 1.706056],accel_mss,speed_ms,0,blend_radius_m)
    movel([0.135106, -1.201803, -2.679250, -0.831336, 1.570796, 1.705902],accel_mss,speed_ms,0,blend_radius_m)
    movel([0.134979, -1.201569, -2.679361, -0.831459, 1.570796, 1.705775],accel_mss,speed_ms,0,blend_radius_m)
    movel([0.135022, -1.201232, -2.679522, -0.831635, 1.570796, 1.705819],accel_mss,speed_ms,0,blend_radius_m)
    movel([0.135228, -1.200845, -2.679706, -0.831838, 1.570796, 1.706025],accel_mss,speed_ms,0,blend_radius_m)
    movel([0.135563, -1.200478, -2.679880, -0.832031, 1.570796, 1.706360],accel_mss,speed_ms,0,blend_radius_m)
    movel([0.136122, -1.200108, -2.680056, -0.832225, 1.570796, 1.706918],accel_mss,speed_ms,0,blend_radius_m)
    movel([0.136520, -1.199894, -2.680158, -0.832338, 1.570796, 1.707316],accel_mss,speed_ms,0,blend_radius_m)
    movel([0.136917, -1.199704, -2.680247, -0.832437, 1.570796, 1.707713],accel_mss,speed_ms,0,blend_radius_m)
    movel([0.137667, -1.199410, -2.680387, -0.832592, 1.570796, 1.708464],accel_mss,speed_ms,0,blend_radius_m)
    movel([0.138053, -1.199378, -2.680402, -0.832609, 1.570796, 1.708850],accel_mss,speed_ms,0,blend_radius_m)
    movel([0.138221, -1.199571, -2.680311, -0.832507, 1.570796, 1.709017],accel_mss,speed_ms,0,blend_radius_m)
    movel([0.138216, -1.200038, -2.680089, -0.832262, 1.570796, 1.709012],accel_mss,speed_ms,0,blend_radius_m)
    movel([0.138152, -1.200373, -2.679930, -0.832086, 1.570796, 1.708948],accel_mss,speed_ms,0,blend_radius_m)
    movel([0.137928, -1.200692, -2.679779, -0.831918, 1.570796, 1.708725],accel_mss,speed_ms,0,blend_radius_m)
    movel([0.137210, -1.201114, -2.679578, -0.831697, 1.570796, 1.708006],accel_mss,speed_ms,0,blend_radius_m)
    movel([0.137030, -1.201442, -2.679422, -0.831525, 1.570796, 1.707826],accel_mss,speed_ms,0,blend_radius_m)
    movel([0.137325, -1.201401, -2.679441, -0.831547, 1.570796, 1.708122],accel_mss,speed_ms,0,blend_radius_m)
    movel([0.137916, -1.201347, -2.679467, -0.831575, 1.570796, 1.708712],accel_mss,speed_ms,0,blend_radius_m)
    movel([0.138103, -1.201603, -2.679345, -0.831441, 1.570796, 1.708899],accel_mss,speed_ms,0,blend_radius_m)
    movel([0.137849, -1.202015, -2.679149, -0.831225, 1.570796, 1.708645],accel_mss,speed_ms,0,blend_radius_m)
    movel([0.137229, -1.202390, -2.678970, -0.831029, 1.570796, 1.708025],accel_mss,speed_ms,0,blend_radius_m)
    movel([0.136800, -1.202622, -2.678859, -0.830908, 1.570796, 1.707596],accel_mss,speed_ms,0,blend_radius_m)
    movel([0.137077, -1.202844, -2.678753, -0.830792, 1.570796, 1.707873],accel_mss,speed_ms,0,blend_radius_m)
    movel([0.137743, -1.202649, -2.678846, -0.830894, 1.570796, 1.708539],accel_mss,speed_ms,0,blend_radius_m)
    movel([0.139062, -1.202207, -2.679057, -0.831125, 1.570796, 1.709859],accel_mss,speed_ms,0,blend_radius_m)
    movel([0.140035, -1.201878, -2.679214, -0.831297, 1.570796, 1.710832],accel_mss,speed_ms,0,blend_radius_m)
    movel([0.140925, -1.201580, -2.679356, -0.831453, 1.570796, 1.711721],accel_mss,speed_ms,0,blend_radius_m)
    movel([0.141673, -1.201328, -2.679476, -0.831585, 1.570796, 1.712470],accel_mss,speed_ms,0,blend_radius_m)
    movel([0.142196, -1.201141, -2.679565, -0.831683, 1.570796, 1.712992],accel_mss,speed_ms,0,blend_radius_m)
    movel([0.142396, -1.200636, -2.679805, -0.831948, 1.570796, 1.713192],accel_mss,speed_ms,0,blend_radius_m)
    movel([0.142482, -1.200188, -2.680018, -0.832183, 1.570796, 1.713278],accel_mss,speed_ms,0,blend_radius_m)
    movel([0.142693, -1.199860, -2.680174, -0.832355, 1.570796, 1.713489],accel_mss,speed_ms,0,blend_radius_m)
    movel([0.143073, -1.199593, -2.680300, -0.832496, 1.570796, 1.713870],accel_mss,speed_ms,0,blend_radius_m)
    movel([0.143726, -1.199329, -2.680426, -0.832635, 1.570796, 1.714522],accel_mss,speed_ms,0,blend_radius_m)
    movel([0.144613, -1.199079, -2.680544, -0.832766, 1.570796, 1.715409],accel_mss,speed_ms,0,blend_radius_m)
    movel([0.146289, -1.198744, -2.680703, -0.832943, 1.570796, 1.717085],accel_mss,speed_ms,0,blend_radius_m)
    movel([0.148054, -1.198438, -2.680847, -0.833104, 1.570796, 1.718850],accel_mss,speed_ms,0,blend_radius_m)
    movel([0.149467, -1.198253, -2.680935, -0.833201, 1.570796, 1.720263],accel_mss,speed_ms,0,blend_radius_m)
    movel([0.150215, -1.198250, -2.680936, -0.833203, 1.570796, 1.721012],accel_mss,speed_ms,0,blend_radius_m)
    movel([0.150569, -1.198467, -2.680833, -0.833088, 1.570796, 1.721365],accel_mss,speed_ms,0,blend_radius_m)
    movel([0.150549, -1.198880, -2.680638, -0.832871, 1.570796, 1.721345],accel_mss,speed_ms,0,blend_radius_m)
    movel([0.150172, -1.199478, -2.680355, -0.832556, 1.570796, 1.720969],accel_mss,speed_ms,0,blend_radius_m)
    movel([0.149950, -1.199809, -2.680198, -0.832382, 1.570796, 1.720746],accel_mss,speed_ms,0,blend_radius_m)
    movel([0.150186, -1.199882, -2.680163, -0.832344, 1.570796, 1.720983],accel_mss,speed_ms,0,blend_radius_m)
    movel([0.151955, -1.199821, -2.680192, -0.832376, 1.570796, 1.722751],accel_mss,speed_ms,0,blend_radius_m)
    movel([0.153640, -1.199750, -2.680226, -0.832413, 1.570796, 1.724436],accel_mss,speed_ms,0,blend_radius_m)
    movel([0.154196, -1.199681, -2.680259, -0.832450, 1.570796, 1.724992],accel_mss,speed_ms,0,blend_radius_m)
    movel([0.154590, -1.199573, -2.680310, -0.832506, 1.570796, 1.725386],accel_mss,speed_ms,0,blend_radius_m)
    movel([0.154444, -1.199201, -2.680486, -0.832702, 1.570796, 1.725241],accel_mss,speed_ms,0,blend_radius_m)
    movel([0.154519, -1.198822, -2.680666, -0.832901, 1.570796, 1.725315],accel_mss,speed_ms,0,blend_radius_m)
    movel([0.154747, -1.198445, -2.680844, -0.833100, 1.570796, 1.725543],accel_mss,speed_ms,0,blend_radius_m)
    movel([0.155058, -1.198208, -2.680956, -0.833225, 1.570796, 1.725854],accel_mss,speed_ms,0,blend_radius_m)
    movel([0.155384, -1.198068, -2.681022, -0.833299, 1.570796, 1.726181],accel_mss,speed_ms,0,blend_radius_m)
    movel([0.155303, -1.197575, -2.681255, -0.833559, 1.570796, 1.726099],accel_mss,speed_ms,0,blend_radius_m)
    movel([0.155399, -1.197207, -2.681429, -0.833754, 1.570796, 1.726195],accel_mss,speed_ms,0,blend_radius_m)
    movel([0.155618, -1.196821, -2.681610, -0.833957, 1.570796, 1.726414],accel_mss,speed_ms,0,blend_radius_m)
    movel([0.155910, -1.196521, -2.681752, -0.834116, 1.570796, 1.726707],accel_mss,speed_ms,0,blend_radius_m)
    movel([0.156578, -1.196229, -2.681889, -0.834271, 1.570796, 1.727375],accel_mss,speed_ms,0,blend_radius_m)
    movel([0.157432, -1.196281, -2.681864, -0.834243, 1.570796, 1.728228],accel_mss,speed_ms,0,blend_radius_m)
    movel([0.158123, -1.196578, -2.681725, -0.834086, 1.570796, 1.728920],accel_mss,speed_ms,0,blend_radius_m)
    movel([0.158279, -1.197056, -2.681500, -0.833834, 1.570796, 1.729075],accel_mss,speed_ms,0,blend_radius_m)
    movel([0.158145, -1.197401, -2.681337, -0.833651, 1.570796, 1.728941],accel_mss,speed_ms,0,blend_radius_m)
    movel([0.157855, -1.197804, -2.681147, -0.833438, 1.570796, 1.728652],accel_mss,speed_ms,0,blend_radius_m)
    movel([0.157522, -1.198122, -2.680996, -0.833270, 1.570796, 1.728318],accel_mss,speed_ms,0,blend_radius_m)
    movel([0.157209, -1.198249, -2.680936, -0.833203, 1.570796, 1.728005],accel_mss,speed_ms,0,blend_radius_m)
    movel([0.157324, -1.198535, -2.680801, -0.833053, 1.570796, 1.728120],accel_mss,speed_ms,0,blend_radius_m)
    movel([0.157482, -1.198741, -2.680704, -0.832944, 1.570796, 1.728278],accel_mss,speed_ms,0,blend_radius_m)
    movel([0.157265, -1.199231, -2.680472, -0.832686, 1.570796, 1.728062],accel_mss,speed_ms,0,blend_radius_m)
    movel([0.156939, -1.199544, -2.680324, -0.832522, 1.570796, 1.727736],accel_mss,speed_ms,0,blend_radius_m)
    movel([0.156605, -1.199765, -2.680219, -0.832405, 1.570796, 1.727401],accel_mss,speed_ms,0,blend_radius_m)
    movel([0.156890, -1.200118, -2.680051, -0.832220, 1.570796, 1.727686],accel_mss,speed_ms,0,blend_radius_m)
    movel([0.157140, -1.200201, -2.680012, -0.832176, 1.570796, 1.727937],accel_mss,speed_ms,0,blend_radius_m)
    movel([0.157374, -1.200299, -2.679965, -0.832125, 1.570796, 1.728170],accel_mss,speed_ms,0,blend_radius_m)
    movel([0.157666, -1.200464, -2.679887, -0.832038, 1.570796, 1.728462],accel_mss,speed_ms,0,blend_radius_m)
    movel([0.157753, -1.200981, -2.679641, -0.831767, 1.570796, 1.728550],accel_mss,speed_ms,0,blend_radius_m)
    movel([0.157631, -1.201345, -2.679468, -0.831576, 1.570796, 1.728427],accel_mss,speed_ms,0,blend_radius_m)
    movel([0.157410, -1.201726, -2.679287, -0.831377, 1.570796, 1.728206],accel_mss,speed_ms,0,blend_radius_m)
    movel([0.157110, -1.202094, -2.679111, -0.831184, 1.570796, 1.727906],accel_mss,speed_ms,0,blend_radius_m)
    movel([0.156493, -1.202431, -2.678950, -0.831008, 1.570796, 1.727289],accel_mss,speed_ms,0,blend_radius_m)
    movel([0.155987, -1.202487, -2.678923, -0.830978, 1.570796, 1.726784],accel_mss,speed_ms,0,blend_radius_m)
    movel([0.155517, -1.202521, -2.678907, -0.830960, 1.570796, 1.726313],accel_mss,speed_ms,0,blend_radius_m)
    movel([0.156081, -1.202850, -2.678750, -0.830789, 1.570796, 1.726877],accel_mss,speed_ms,0,blend_radius_m)
    movel([0.156250, -1.203378, -2.678498, -0.830513, 1.570796, 1.727047],accel_mss,speed_ms,0,blend_radius_m)
    movel([0.156200, -1.204426, -2.677996, -0.829967, 1.570796, 1.726996],accel_mss,speed_ms,0,blend_radius_m)
    movel([0.155879, -1.206537, -2.676981, -0.828871, 1.570796, 1.726675],accel_mss,speed_ms,0,blend_radius_m)
    movel([0.155597, -1.208137, -2.676209, -0.828043, 1.570796, 1.726393],accel_mss,speed_ms,0,blend_radius_m)
    movel([0.155343, -1.209346, -2.675624, -0.827420, 1.570796, 1.726140],accel_mss,speed_ms,0,blend_radius_m)
    movel([0.155059, -1.210462, -2.675082, -0.826846, 1.570796, 1.725856],accel_mss,speed_ms,0,blend_radius_m)
    movel([0.154680, -1.211740, -2.674459, -0.826190, 1.570796, 1.725476],accel_mss,speed_ms,0,blend_radius_m)
    movel([0.153984, -1.213905, -2.673401, -0.825083, 1.570796, 1.724781],accel_mss,speed_ms,0,blend_radius_m)
    movel([0.153418, -1.215525, -2.672605, -0.824258, 1.570796, 1.724214],accel_mss,speed_ms,0,blend_radius_m)
    movel([0.152953, -1.216731, -2.672011, -0.823646, 1.570796, 1.723749],accel_mss,speed_ms,0,blend_radius_m)
    movel([0.152673, -1.217179, -2.671790, -0.823420, 1.570796, 1.723469],accel_mss,speed_ms,0,blend_radius_m)
    movel([0.152497, -1.217483, -2.671640, -0.823266, 1.570796, 1.723293],accel_mss,speed_ms,0,blend_radius_m)
    movel([0.152728, -1.217731, -2.671518, -0.823141, 1.570796, 1.723524],accel_mss,speed_ms,0,blend_radius_m)
    movel([0.152948, -1.217958, -2.671405, -0.823026, 1.570796, 1.723744],accel_mss,speed_ms,0,blend_radius_m)
    movel([0.152699, -1.218550, -2.671112, -0.822727, 1.570796, 1.723495],accel_mss,speed_ms,0,blend_radius_m)
    movel([0.151831, -1.218842, -2.670968, -0.822579, 1.570796, 1.722627],accel_mss,speed_ms,0,blend_radius_m)
    movel([0.150034, -1.219185, -2.670797, -0.822406, 1.570796, 1.720831],accel_mss,speed_ms,0,blend_radius_m)
    movel([0.144850, -1.220010, -2.670388, -0.821991, 1.570796, 1.715647],accel_mss,speed_ms,0,blend_radius_m)
    movel([0.137167, -1.221258, -2.669767, -0.821364, 1.570796, 1.707964],accel_mss,speed_ms,0,blend_radius_m)
    speed_ms = 0.003
    movel([0.137167, -1.206848, -2.662674, -0.842866, 1.570796, 1.707964],accel_mss,speed_ms,0,blend_radius_m)
    speed_ms = 1.000
    movel([0.137167, -1.179616, -2.648120, -0.884653, 1.570796, 1.707964],accel_mss,speed_ms,0,blend_radius_m)
    movel([0.151082, -1.164224, -2.655255, -0.892909, 1.570796, 1.721879],accel_mss,speed_ms,0,blend_radius_m)
    movel([0.151082, -1.191573, -2.670012, -0.850804, 1.570796, 1.721879],accel_mss,speed_ms,0,blend_radius_m)
    speed_ms = 0.003
    movel([0.151082, -1.202391, -2.675421, -0.834578, 1.570796, 1.721879],accel_mss,speed_ms,0,blend_radius_m)
    speed_ms = 0.007
    movel([0.150969, -1.202053, -2.675582, -0.834754, 1.570796, 1.721765],accel_mss,speed_ms,0,blend_radius_m)
    movel([0.151469, -1.201901, -2.675655, -0.834833, 1.570796, 1.722265],accel_mss,speed_ms,0,blend_radius_m)
    movel([0.151953, -1.201863, -2.675673, -0.834852, 1.570796, 1.722750],accel_mss,speed_ms,0,blend_radius_m)
    movel([0.152627, -1.201852, -2.675678, -0.834858, 1.570796, 1.723424],accel_mss,speed_ms,0,blend_radius_m)
    movel([0.153372, -1.201867, -2.675671, -0.834851, 1.570796, 1.724169],accel_mss,speed_ms,0,blend_radius_m)
    movel([0.153785, -1.201912, -2.675650, -0.834827, 1.570796, 1.724581],accel_mss,speed_ms,0,blend_radius_m)
    movel([0.154057, -1.202126, -2.675547, -0.834715, 1.570796, 1.724853],accel_mss,speed_ms,0,blend_radius_m)
    movel([0.153797, -1.202439, -2.675398, -0.834552, 1.570796, 1.724593],accel_mss,speed_ms,0,blend_radius_m)
    movel([0.153457, -1.202479, -2.675379, -0.834532, 1.570796, 1.724253],accel_mss,speed_ms,0,blend_radius_m)
    movel([0.152457, -1.202484, -2.675376, -0.834529, 1.570796, 1.723254],accel_mss,speed_ms,0,blend_radius_m)
    movel([0.151560, -1.202464, -2.675386, -0.834539, 1.570796, 1.722356],accel_mss,speed_ms,0,blend_radius_m)
    movel([0.151082, -1.202391, -2.675421, -0.834578, 1.570796, 1.721879],accel_mss,speed_ms,0,blend_radius_m)
    speed_ms = 0.003
    movel([0.151082, -1.206066, -2.677208, -0.829115, 1.570796, 1.721879],accel_mss,speed_ms,0,blend_radius_m)
    speed_ms = 0.007
    movel([0.150969, -1.205729, -2.677370, -0.829290, 1.570796, 1.721765],accel_mss,speed_ms,0,blend_radius_m)
    movel([0.151469, -1.205577, -2.677443, -0.829368, 1.570796, 1.722265],accel_mss,speed_ms,0,blend_radius_m)
    movel([0.151953, -1.205540, -2.677461, -0.829388, 1.570796, 1.722750],accel_mss,speed_ms,0,blend_radius_m)
    movel([0.152627, -1.205529, -2.677466, -0.829394, 1.570796, 1.723424],accel_mss,speed_ms,0,blend_radius_m)
    movel([0.153372, -1.205543, -2.677459, -0.829386, 1.570796, 1.724169],accel_mss,speed_ms,0,blend_radius_m)
    movel([0.153785, -1.205588, -2.677438, -0.829363, 1.570796, 1.724581],accel_mss,speed_ms,0,blend_radius_m)
    movel([0.154057, -1.205802, -2.677335, -0.829252, 1.570796, 1.724853],accel_mss,speed_ms,0,blend_radius_m)
    movel([0.153797, -1.206114, -2.677185, -0.829090, 1.570796, 1.724593],accel_mss,speed_ms,0,blend_radius_m)
    movel([0.153457, -1.206154, -2.677166, -0.829069, 1.570796, 1.724253],accel_mss,speed_ms,0,blend_radius_m)
    movel([0.152457, -1.206160, -2.677163, -0.829066, 1.570796, 1.723254],accel_mss,speed_ms,0,blend_radius_m)
    movel([0.151560, -1.206140, -2.677173, -0.829077, 1.570796, 1.722356],accel_mss,speed_ms,0,blend_radius_m)
    movel([0.151082, -1.206066, -2.677208, -0.829115, 1.570796, 1.721879],accel_mss,speed_ms,0,blend_radius_m)
    speed_ms = 0.003
    movel([0.151082, -1.191573, -2.670012, -0.850804, 1.570796, 1.721879],accel_mss,speed_ms,0,blend_radius_m)
    speed_ms = 1.000
    movel([0.151082, -1.164224, -2.655255, -0.892909, 1.570796, 1.721879],accel_mss,speed_ms,0,blend_radius_m)
    movel([0.145352, -1.167552, -2.653734, -0.891104, 1.570796, 1.716149],accel_mss,speed_ms,0,blend_radius_m)
    movel([0.145352, -1.194877, -2.668447, -0.849065, 1.570796, 1.716149],accel_mss,speed_ms,0,blend_radius_m)
    speed_ms = 0.003
    movel([0.145352, -1.205682, -2.673839, -0.832868, 1.570796, 1.716149],accel_mss,speed_ms,0,blend_radius_m)
    speed_ms = 0.007
    movel([0.144892, -1.206441, -2.673472, -0.832476, 1.570796, 1.715689],accel_mss,speed_ms,0,blend_radius_m)
    movel([0.144137, -1.207398, -2.673009, -0.831982, 1.570796, 1.714933],accel_mss,speed_ms,0,blend_radius_m)
    movel([0.143636, -1.208021, -2.672707, -0.831661, 1.570796, 1.714432],accel_mss,speed_ms,0,blend_radius_m)
    movel([0.143137, -1.208649, -2.672402, -0.831338, 1.570796, 1.713934],accel_mss,speed_ms,0,blend_radius_m)
    movel([0.142703, -1.209200, -2.672134, -0.831055, 1.570796, 1.713499],accel_mss,speed_ms,0,blend_radius_m)
    movel([0.142437, -1.209541, -2.671968, -0.830880, 1.570796, 1.713233],accel_mss,speed_ms,0,blend_radius_m)
    movel([0.142176, -1.209872, -2.671807, -0.830710, 1.570796, 1.712972],accel_mss,speed_ms,0,blend_radius_m)
    movel([0.141758, -1.210380, -2.671559, -0.830450, 1.570796, 1.712554],accel_mss,speed_ms,0,blend_radius_m)
    movel([0.141285, -1.210949, -2.671282, -0.830159, 1.570796, 1.712081],accel_mss,speed_ms,0,blend_radius_m)
    movel([0.140814, -1.211503, -2.671011, -0.829875, 1.570796, 1.711611],accel_mss,speed_ms,0,blend_radius_m)
    movel([0.140259, -1.212142, -2.670698, -0.829549, 1.570796, 1.711056],accel_mss,speed_ms,0,blend_radius_m)
    movel([0.139901, -1.212511, -2.670517, -0.829361, 1.570796, 1.710698],accel_mss,speed_ms,0,blend_radius_m)
    movel([0.139535, -1.212726, -2.670412, -0.829251, 1.570796, 1.710331],accel_mss,speed_ms,0,blend_radius_m)
    movel([0.139579, -1.212376, -2.670583, -0.829429, 1.570796, 1.710375],accel_mss,speed_ms,0,blend_radius_m)
    movel([0.139763, -1.211998, -2.670769, -0.829623, 1.570796, 1.710559],accel_mss,speed_ms,0,blend_radius_m)
    movel([0.140108, -1.211392, -2.671065, -0.829932, 1.570796, 1.710904],accel_mss,speed_ms,0,blend_radius_m)
    movel([0.140407, -1.210885, -2.671313, -0.830191, 1.570796, 1.711203],accel_mss,speed_ms,0,blend_radius_m)
    movel([0.140707, -1.210391, -2.671554, -0.830444, 1.570796, 1.711503],accel_mss,speed_ms,0,blend_radius_m)
    movel([0.140974, -1.209961, -2.671764, -0.830665, 1.570796, 1.711770],accel_mss,speed_ms,0,blend_radius_m)
    movel([0.141294, -1.209489, -2.671994, -0.830907, 1.570796, 1.712090],accel_mss,speed_ms,0,blend_radius_m)
    movel([0.141511, -1.209164, -2.672151, -0.831073, 1.570796, 1.712307],accel_mss,speed_ms,0,blend_radius_m)
    movel([0.141745, -1.208807, -2.672325, -0.831257, 1.570796, 1.712541],accel_mss,speed_ms,0,blend_radius_m)
    movel([0.141961, -1.208467, -2.672490, -0.831432, 1.570796, 1.712758],accel_mss,speed_ms,0,blend_radius_m)
    movel([0.142257, -1.207989, -2.672723, -0.831678, 1.570796, 1.713053],accel_mss,speed_ms,0,blend_radius_m)
    movel([0.142358, -1.207630, -2.672896, -0.831862, 1.570796, 1.713155],accel_mss,speed_ms,0,blend_radius_m)
    movel([0.142144, -1.207479, -2.672969, -0.831940, 1.570796, 1.712941],accel_mss,speed_ms,0,blend_radius_m)
    movel([0.141717, -1.207512, -2.672954, -0.831923, 1.570796, 1.712514],accel_mss,speed_ms,0,blend_radius_m)
    movel([0.140967, -1.207731, -2.672848, -0.831811, 1.570796, 1.711763],accel_mss,speed_ms,0,blend_radius_m)
    movel([0.140661, -1.207762, -2.672832, -0.831794, 1.570796, 1.711458],accel_mss,speed_ms,0,blend_radius_m)
    movel([0.140473, -1.207500, -2.672959, -0.831929, 1.570796, 1.711269],accel_mss,speed_ms,0,blend_radius_m)
    movel([0.140699, -1.206886, -2.673257, -0.832246, 1.570796, 1.711495],accel_mss,speed_ms,0,blend_radius_m)
    movel([0.141722, -1.205147, -2.674096, -0.833145, 1.570796, 1.712519],accel_mss,speed_ms,0,blend_radius_m)
    movel([0.142819, -1.203366, -2.674953, -0.834070, 1.570796, 1.713616],accel_mss,speed_ms,0,blend_radius_m)
    movel([0.143193, -1.202997, -2.675130, -0.834262, 1.570796, 1.713989],accel_mss,speed_ms,0,blend_radius_m)
    movel([0.143687, -1.202784, -2.675233, -0.834373, 1.570796, 1.714484],accel_mss,speed_ms,0,blend_radius_m)
    movel([0.144594, -1.202593, -2.675324, -0.834472, 1.570796, 1.715390],accel_mss,speed_ms,0,blend_radius_m)
    movel([0.145488, -1.202461, -2.675387, -0.834541, 1.570796, 1.716285],accel_mss,speed_ms,0,blend_radius_m)
    movel([0.145650, -1.202689, -2.675278, -0.834422, 1.570796, 1.716446],accel_mss,speed_ms,0,blend_radius_m)
    movel([0.145410, -1.203069, -2.675096, -0.834224, 1.570796, 1.716207],accel_mss,speed_ms,0,blend_radius_m)
    movel([0.145095, -1.203530, -2.674874, -0.833985, 1.570796, 1.715891],accel_mss,speed_ms,0,blend_radius_m)
    movel([0.144710, -1.204047, -2.674626, -0.833716, 1.570796, 1.715506],accel_mss,speed_ms,0,blend_radius_m)
    movel([0.144317, -1.204561, -2.674379, -0.833449, 1.570796, 1.715113],accel_mss,speed_ms,0,blend_radius_m)
    movel([0.143987, -1.205009, -2.674163, -0.833217, 1.570796, 1.714783],accel_mss,speed_ms,0,blend_radius_m)
    movel([0.143713, -1.205390, -2.673980, -0.833020, 1.570796, 1.714510],accel_mss,speed_ms,0,blend_radius_m)
    movel([0.143899, -1.205667, -2.673846, -0.832876, 1.570796, 1.714695],accel_mss,speed_ms,0,blend_radius_m)
    movel([0.144192, -1.205681, -2.673839, -0.832869, 1.570796, 1.714988],accel_mss,speed_ms,0,blend_radius_m)
    movel([0.144594, -1.205631, -2.673863, -0.832895, 1.570796, 1.715390],accel_mss,speed_ms,0,blend_radius_m)
    movel([0.145044, -1.205565, -2.673895, -0.832929, 1.570796, 1.715840],accel_mss,speed_ms,0,blend_radius_m)
    movel([0.145352, -1.205682, -2.673839, -0.832868, 1.570796, 1.716149],accel_mss,speed_ms,0,blend_radius_m)
    speed_ms = 0.003
    movel([0.145352, -1.209353, -2.675620, -0.827416, 1.570796, 1.716149],accel_mss,speed_ms,0,blend_radius_m)
    speed_ms = 0.007
    movel([0.144892, -1.210111, -2.675252, -0.827026, 1.570796, 1.715689],accel_mss,speed_ms,0,blend_radius_m)
    movel([0.144137, -1.211066, -2.674788, -0.826535, 1.570796, 1.714933],accel_mss,speed_ms,0,blend_radius_m)
    movel([0.143636, -1.211689, -2.674484, -0.826216, 1.570796, 1.714432],accel_mss,speed_ms,0,blend_radius_m)
    movel([0.143137, -1.212315, -2.674178, -0.825895, 1.570796, 1.713934],accel_mss,speed_ms,0,blend_radius_m)
    movel([0.142703, -1.212866, -2.673909, -0.825613, 1.570796, 1.713499],accel_mss,speed_ms,0,blend_radius_m)
    movel([0.142437, -1.213206, -2.673743, -0.825440, 1.570796, 1.713233],accel_mss,speed_ms,0,blend_radius_m)
    movel([0.142176, -1.213537, -2.673581, -0.825271, 1.570796, 1.712972],accel_mss,speed_ms,0,blend_radius_m)
    movel([0.141758, -1.214044, -2.673333, -0.825012, 1.570796, 1.712554],accel_mss,speed_ms,0,blend_radius_m)
    movel([0.141285, -1.214612, -2.673054, -0.824723, 1.570796, 1.712081],accel_mss,speed_ms,0,blend_radius_m)
    movel([0.140814, -1.215166, -2.672782, -0.824441, 1.570796, 1.711611],accel_mss,speed_ms,0,blend_radius_m)
    movel([0.140259, -1.215804, -2.672468, -0.824117, 1.570796, 1.711056],accel_mss,speed_ms,0,blend_radius_m)
    movel([0.139901, -1.216171, -2.672287, -0.823930, 1.570796, 1.710698],accel_mss,speed_ms,0,blend_radius_m)
    movel([0.139535, -1.216387, -2.672181, -0.823821, 1.570796, 1.710331],accel_mss,speed_ms,0,blend_radius_m)
    movel([0.139579, -1.216037, -2.672353, -0.823998, 1.570796, 1.710375],accel_mss,speed_ms,0,blend_radius_m)
    movel([0.139763, -1.215659, -2.672540, -0.824190, 1.570796, 1.710559],accel_mss,speed_ms,0,blend_radius_m)
    movel([0.140108, -1.215054, -2.672837, -0.824498, 1.570796, 1.710904],accel_mss,speed_ms,0,blend_radius_m)
    movel([0.140407, -1.214548, -2.673085, -0.824755, 1.570796, 1.711203],accel_mss,speed_ms,0,blend_radius_m)
    movel([0.140707, -1.214055, -2.673328, -0.825007, 1.570796, 1.711503],accel_mss,speed_ms,0,blend_radius_m)
    movel([0.140974, -1.213625, -2.673538, -0.825226, 1.570796, 1.711770],accel_mss,speed_ms,0,blend_radius_m)
    movel([0.141294, -1.213154, -2.673769, -0.825466, 1.570796, 1.712090],accel_mss,speed_ms,0,blend_radius_m)
    movel([0.141511, -1.212830, -2.673927, -0.825632, 1.570796, 1.712307],accel_mss,speed_ms,0,blend_radius_m)
    movel([0.141745, -1.212474, -2.674101, -0.825814, 1.570796, 1.712541],accel_mss,speed_ms,0,blend_radius_m)
    movel([0.141961, -1.212134, -2.674267, -0.825988, 1.570796, 1.712758],accel_mss,speed_ms,0,blend_radius_m)
    movel([0.142257, -1.211656, -2.674500, -0.826233, 1.570796, 1.713053],accel_mss,speed_ms,0,blend_radius_m)
    movel([0.142358, -1.211298, -2.674674, -0.826416, 1.570796, 1.713155],accel_mss,speed_ms,0,blend_radius_m)
    movel([0.142144, -1.211148, -2.674748, -0.826493, 1.570796, 1.712941],accel_mss,speed_ms,0,blend_radius_m)
    movel([0.141717, -1.211180, -2.674732, -0.826477, 1.570796, 1.712514],accel_mss,speed_ms,0,blend_radius_m)
    movel([0.140967, -1.211398, -2.674626, -0.826365, 1.570796, 1.711763],accel_mss,speed_ms,0,blend_radius_m)
    movel([0.140661, -1.211430, -2.674610, -0.826349, 1.570796, 1.711458],accel_mss,speed_ms,0,blend_radius_m)
    movel([0.140473, -1.211169, -2.674738, -0.826483, 1.570796, 1.711269],accel_mss,speed_ms,0,blend_radius_m)
    movel([0.140699, -1.210555, -2.675036, -0.826798, 1.570796, 1.711495],accel_mss,speed_ms,0,blend_radius_m)
    movel([0.141722, -1.208819, -2.675879, -0.827691, 1.570796, 1.712519],accel_mss,speed_ms,0,blend_radius_m)
    movel([0.142819, -1.207041, -2.676738, -0.828610, 1.570796, 1.713616],accel_mss,speed_ms,0,blend_radius_m)
    movel([0.143193, -1.206671, -2.676917, -0.828801, 1.570796, 1.713989],accel_mss,speed_ms,0,blend_radius_m)
    movel([0.143687, -1.206459, -2.677019, -0.828911, 1.570796, 1.714484],accel_mss,speed_ms,0,blend_radius_m)
    movel([0.144594, -1.206268, -2.677111, -0.829010, 1.570796, 1.715390],accel_mss,speed_ms,0,blend_radius_m)
    movel([0.145488, -1.206137, -2.677174, -0.829078, 1.570796, 1.716285],accel_mss,speed_ms,0,blend_radius_m)
    movel([0.145650, -1.206364, -2.677065, -0.828960, 1.570796, 1.716446],accel_mss,speed_ms,0,blend_radius_m)
    movel([0.145410, -1.206744, -2.676882, -0.828763, 1.570796, 1.716207],accel_mss,speed_ms,0,blend_radius_m)
    movel([0.145095, -1.207204, -2.676660, -0.828525, 1.570796, 1.715891],accel_mss,speed_ms,0,blend_radius_m)
    movel([0.144710, -1.207720, -2.676410, -0.828258, 1.570796, 1.715506],accel_mss,speed_ms,0,blend_radius_m)
    movel([0.144317, -1.208233, -2.676162, -0.827993, 1.570796, 1.715113],accel_mss,speed_ms,0,blend_radius_m)
    movel([0.143987, -1.208681, -2.675946, -0.827762, 1.570796, 1.714783],accel_mss,speed_ms,0,blend_radius_m)
    movel([0.143713, -1.209061, -2.675762, -0.827566, 1.570796, 1.714510],accel_mss,speed_ms,0,blend_radius_m)
    movel([0.143899, -1.209338, -2.675627, -0.827423, 1.570796, 1.714695],accel_mss,speed_ms,0,blend_radius_m)
    movel([0.144192, -1.209352, -2.675620, -0.827416, 1.570796, 1.714988],accel_mss,speed_ms,0,blend_radius_m)
    movel([0.144594, -1.209302, -2.675645, -0.827442, 1.570796, 1.715390],accel_mss,speed_ms,0,blend_radius_m)
    movel([0.145044, -1.209236, -2.675677, -0.827476, 1.570796, 1.715840],accel_mss,speed_ms,0,blend_radius_m)
    movel([0.145352, -1.209353, -2.675620, -0.827416, 1.570796, 1.716149],accel_mss,speed_ms,0,blend_radius_m)
    speed_ms = 0.003
    movel([0.145352, -1.194877, -2.668447, -0.849065, 1.570796, 1.716149],accel_mss,speed_ms,0,blend_radius_m)
    speed_ms = 1.000
    movel([0.145352, -1.167552, -2.653734, -0.891104, 1.570796, 1.716149],accel_mss,speed_ms,0,blend_radius_m)
    movel([0.137055, -1.166453, -2.654237, -0.891698, 1.570796, 1.707851],accel_mss,speed_ms,0,blend_radius_m)
    movel([0.137055, -1.193786, -2.668965, -0.849638, 1.570796, 1.707851],accel_mss,speed_ms,0,blend_radius_m)
    speed_ms = 0.003
    movel([0.137055, -1.204595, -2.674362, -0.833431, 1.570796, 1.707851],accel_mss,speed_ms,0,blend_radius_m)
    speed_ms = 0.007
    movel([0.136494, -1.204950, -2.674191, -0.833247, 1.570796, 1.707290],accel_mss,speed_ms,0,blend_radius_m)
    movel([0.136049, -1.205173, -2.674084, -0.833132, 1.570796, 1.706845],accel_mss,speed_ms,0,blend_radius_m)
    movel([0.135574, -1.205676, -2.673841, -0.832872, 1.570796, 1.706370],accel_mss,speed_ms,0,blend_radius_m)
    movel([0.135443, -1.206057, -2.673658, -0.832675, 1.570796, 1.706239],accel_mss,speed_ms,0,blend_radius_m)
    movel([0.135291, -1.206439, -2.673473, -0.832477, 1.570796, 1.706087],accel_mss,speed_ms,0,blend_radius_m)
    movel([0.134927, -1.206706, -2.673344, -0.832339, 1.570796, 1.705723],accel_mss,speed_ms,0,blend_radius_m)
    movel([0.134854, -1.206313, -2.673534, -0.832542, 1.570796, 1.705650],accel_mss,speed_ms,0,blend_radius_m)
    movel([0.134864, -1.205964, -2.673703, -0.832723, 1.570796, 1.705661],accel_mss,speed_ms,0,blend_radius_m)
    movel([0.134522, -1.205699, -2.673830, -0.832859, 1.570796, 1.705319],accel_mss,speed_ms,0,blend_radius_m)
    movel([0.134069, -1.205720, -2.673820, -0.832849, 1.570796, 1.704865],accel_mss,speed_ms,0,blend_radius_m)
    movel([0.133654, -1.205719, -2.673821, -0.832849, 1.570796, 1.704450],accel_mss,speed_ms,0,blend_radius_m)
    movel([0.133786, -1.205330, -2.674009, -0.833051, 1.570796, 1.704582],accel_mss,speed_ms,0,blend_radius_m)
    movel([0.134311, -1.205057, -2.674140, -0.833192, 1.570796, 1.705107],accel_mss,speed_ms,0,blend_radius_m)
    movel([0.134751, -1.204849, -2.674240, -0.833300, 1.570796, 1.705547],accel_mss,speed_ms,0,blend_radius_m)
    movel([0.135054, -1.204524, -2.674397, -0.833469, 1.570796, 1.705850],accel_mss,speed_ms,0,blend_radius_m)
    movel([0.135170, -1.204147, -2.674578, -0.833664, 1.570796, 1.705966],accel_mss,speed_ms,0,blend_radius_m)
    movel([0.135357, -1.203662, -2.674811, -0.833916, 1.570796, 1.706154],accel_mss,speed_ms,0,blend_radius_m)
    movel([0.135738, -1.203369, -2.674952, -0.834068, 1.570796, 1.706534],accel_mss,speed_ms,0,blend_radius_m)
    movel([0.135799, -1.203822, -2.674734, -0.833833, 1.570796, 1.706596],accel_mss,speed_ms,0,blend_radius_m)
    movel([0.135779, -1.204238, -2.674534, -0.833617, 1.570796, 1.706575],accel_mss,speed_ms,0,blend_radius_m)
    movel([0.135884, -1.204456, -2.674429, -0.833504, 1.570796, 1.706680],accel_mss,speed_ms,0,blend_radius_m)
    movel([0.136517, -1.204422, -2.674445, -0.833521, 1.570796, 1.707313],accel_mss,speed_ms,0,blend_radius_m)
    movel([0.136880, -1.204323, -2.674493, -0.833573, 1.570796, 1.707676],accel_mss,speed_ms,0,blend_radius_m)
    movel([0.137133, -1.204438, -2.674438, -0.833513, 1.570796, 1.707930],accel_mss,speed_ms,0,blend_radius_m)
    speed_ms = 0.003
    movel([0.137055, -1.208268, -2.676146, -0.827975, 1.570796, 1.707851],accel_mss,speed_ms,0,blend_radius_m)
    speed_ms = 0.007
    movel([0.136494, -1.208622, -2.675974, -0.827793, 1.570796, 1.707290],accel_mss,speed_ms,0,blend_radius_m)
    movel([0.136049, -1.208844, -2.675867, -0.827678, 1.570796, 1.706845],accel_mss,speed_ms,0,blend_radius_m)
    movel([0.135574, -1.209347, -2.675623, -0.827419, 1.570796, 1.706370],accel_mss,speed_ms,0,blend_radius_m)
    movel([0.135443, -1.209727, -2.675439, -0.827223, 1.570796, 1.706239],accel_mss,speed_ms,0,blend_radius_m)
    movel([0.135291, -1.210109, -2.675253, -0.827027, 1.570796, 1.706087],accel_mss,speed_ms,0,blend_radius_m)
    movel([0.134927, -1.210376, -2.675124, -0.826890, 1.570796, 1.705723],accel_mss,speed_ms,0,blend_radius_m)
    movel([0.134854, -1.209983, -2.675314, -0.827092, 1.570796, 1.705650],accel_mss,speed_ms,0,blend_radius_m)
    movel([0.134864, -1.209634, -2.675484, -0.827271, 1.570796, 1.705661],accel_mss,speed_ms,0,blend_radius_m)
    movel([0.134522, -1.209370, -2.675612, -0.827407, 1.570796, 1.705319],accel_mss,speed_ms,0,blend_radius_m)
    movel([0.134069, -1.209391, -2.675602, -0.827397, 1.570796, 1.704865],accel_mss,speed_ms,0,blend_radius_m)
    movel([0.133654, -1.209390, -2.675602, -0.827397, 1.570796, 1.704450],accel_mss,speed_ms,0,blend_radius_m)
    movel([0.133786, -1.209001, -2.675791, -0.827597, 1.570796, 1.704582],accel_mss,speed_ms,0,blend_radius_m)
    movel([0.134311, -1.208729, -2.675923, -0.827738, 1.570796, 1.705107],accel_mss,speed_ms,0,blend_radius_m)
    movel([0.134751, -1.208521, -2.676023, -0.827845, 1.570796, 1.705547],accel_mss,speed_ms,0,blend_radius_m)
    movel([0.135054, -1.208196, -2.676180, -0.828012, 1.570796, 1.705850],accel_mss,speed_ms,0,blend_radius_m)
    movel([0.135170, -1.207820, -2.676362, -0.828207, 1.570796, 1.705966],accel_mss,speed_ms,0,blend_radius_m)
    movel([0.135357, -1.207335, -2.676596, -0.828457, 1.570796, 1.706154],accel_mss,speed_ms,0,blend_radius_m)
    movel([0.135738, -1.207043, -2.676737, -0.828609, 1.570796, 1.706534],accel_mss,speed_ms,0,blend_radius_m)
    movel([0.135799, -1.207495, -2.676519, -0.828375, 1.570796, 1.706596],accel_mss,speed_ms,0,blend_radius_m)
    movel([0.135779, -1.207911, -2.676318, -0.828160, 1.570796, 1.706575],accel_mss,speed_ms,0,blend_radius_m)
    movel([0.135884, -1.208129, -2.676213, -0.828047, 1.570796, 1.706680],accel_mss,speed_ms,0,blend_radius_m)
    movel([0.136517, -1.208095, -2.676229, -0.828065, 1.570796, 1.707313],accel_mss,speed_ms,0,blend_radius_m)
    movel([0.136880, -1.207996, -2.676277, -0.828116, 1.570796, 1.707676],accel_mss,speed_ms,0,blend_radius_m)
    movel([0.137133, -1.208111, -2.676222, -0.828057, 1.570796, 1.707930],accel_mss,speed_ms,0,blend_radius_m)
    speed_ms = 0.003
    movel([0.137055, -1.193786, -2.668965, -0.849638, 1.570796, 1.707851],accel_mss,speed_ms,0,blend_radius_m)
    speed_ms = 1.000
    movel([0.137055, -1.166453, -2.654237, -0.891698, 1.570796, 1.707851],accel_mss,speed_ms,0,blend_radius_m)
    movel([0.143132, -1.157119, -2.658467, -0.896803, 1.570796, 1.713928],accel_mss,speed_ms,0,blend_radius_m)
    movel([0.143132, -1.184515, -2.673317, -0.854557, 1.570796, 1.713928],accel_mss,speed_ms,0,blend_radius_m)
    speed_ms = 0.003
    movel([0.143132, -1.195359, -2.678761, -0.838269, 1.570796, 1.713928],accel_mss,speed_ms,0,blend_radius_m)
    speed_ms = 0.007
    movel([0.143036, -1.195087, -2.678889, -0.838413, 1.570796, 1.713832],accel_mss,speed_ms,0,blend_radius_m)
    movel([0.143116, -1.194584, -2.679126, -0.838679, 1.570796, 1.713912],accel_mss,speed_ms,0,blend_radius_m)
    movel([0.143455, -1.193390, -2.679687, -0.839312, 1.570796, 1.714251],accel_mss,speed_ms,0,blend_radius_m)
    movel([0.144038, -1.192312, -2.680192, -0.839885, 1.570796, 1.714834],accel_mss,speed_ms,0,blend_radius_m)
    movel([0.144785, -1.191486, -2.680578, -0.840325, 1.570796, 1.715582],accel_mss,speed_ms,0,blend_radius_m)
    movel([0.145608, -1.190994, -2.680807, -0.840587, 1.570796, 1.716404],accel_mss,speed_ms,0,blend_radius_m)
    movel([0.146854, -1.190657, -2.680965, -0.840767, 1.570796, 1.717650],accel_mss,speed_ms,0,blend_radius_m)
    movel([0.148797, -1.190334, -2.681115, -0.840940, 1.570796, 1.719593],accel_mss,speed_ms,0,blend_radius_m)
    movel([0.150703, -1.190094, -2.681227, -0.841068, 1.570796, 1.721499],accel_mss,speed_ms,0,blend_radius_m)
    movel([0.151445, -1.190152, -2.681200, -0.841037, 1.570796, 1.722241],accel_mss,speed_ms,0,blend_radius_m)
    movel([0.151684, -1.190327, -2.681118, -0.840944, 1.570796, 1.722480],accel_mss,speed_ms,0,blend_radius_m)
    movel([0.151798, -1.190617, -2.680983, -0.840789, 1.570796, 1.722594],accel_mss,speed_ms,0,blend_radius_m)
    movel([0.151826, -1.190915, -2.680844, -0.840630, 1.570796, 1.722622],accel_mss,speed_ms,0,blend_radius_m)
    movel([0.151840, -1.191333, -2.680649, -0.840406, 1.570796, 1.722636],accel_mss,speed_ms,0,blend_radius_m)
    movel([0.151696, -1.191881, -2.680394, -0.840115, 1.570796, 1.722492],accel_mss,speed_ms,0,blend_radius_m)
    movel([0.151501, -1.192502, -2.680103, -0.839784, 1.570796, 1.722298],accel_mss,speed_ms,0,blend_radius_m)
    movel([0.151280, -1.193108, -2.679819, -0.839462, 1.570796, 1.722077],accel_mss,speed_ms,0,blend_radius_m)
    movel([0.151065, -1.193606, -2.679585, -0.839198, 1.570796, 1.721862],accel_mss,speed_ms,0,blend_radius_m)
    movel([0.150862, -1.193943, -2.679427, -0.839019, 1.570796, 1.721658],accel_mss,speed_ms,0,blend_radius_m)
    movel([0.150403, -1.194304, -2.679258, -0.838828, 1.570796, 1.721200],accel_mss,speed_ms,0,blend_radius_m)
    movel([0.150113, -1.194307, -2.679256, -0.838826, 1.570796, 1.720910],accel_mss,speed_ms,0,blend_radius_m)
    movel([0.149973, -1.194104, -2.679352, -0.838933, 1.570796, 1.720770],accel_mss,speed_ms,0,blend_radius_m)
    movel([0.150015, -1.193666, -2.679557, -0.839166, 1.570796, 1.720811],accel_mss,speed_ms,0,blend_radius_m)
    movel([0.150240, -1.192993, -2.679873, -0.839523, 1.570796, 1.721036],accel_mss,speed_ms,0,blend_radius_m)
    movel([0.150449, -1.192438, -2.680133, -0.839818, 1.570796, 1.721245],accel_mss,speed_ms,0,blend_radius_m)
    movel([0.150527, -1.191917, -2.680377, -0.840096, 1.570796, 1.721323],accel_mss,speed_ms,0,blend_radius_m)
    movel([0.150292, -1.191461, -2.680589, -0.840338, 1.570796, 1.721089],accel_mss,speed_ms,0,blend_radius_m)
    movel([0.150080, -1.191357, -2.680638, -0.840394, 1.570796, 1.720876],accel_mss,speed_ms,0,blend_radius_m)
    movel([0.149720, -1.191338, -2.680647, -0.840404, 1.570796, 1.720516],accel_mss,speed_ms,0,blend_radius_m)
    movel([0.148947, -1.191400, -2.680618, -0.840371, 1.570796, 1.719743],accel_mss,speed_ms,0,blend_radius_m)
    movel([0.147888, -1.191545, -2.680550, -0.840294, 1.570796, 1.718685],accel_mss,speed_ms,0,blend_radius_m)
    movel([0.146788, -1.191786, -2.680438, -0.840166, 1.570796, 1.717584],accel_mss,speed_ms,0,blend_radius_m)
    movel([0.145823, -1.192063, -2.680308, -0.840018, 1.570796, 1.716619],accel_mss,speed_ms,0,blend_radius_m)
    movel([0.145331, -1.192319, -2.680188, -0.839881, 1.570796, 1.716127],accel_mss,speed_ms,0,blend_radius_m)
    movel([0.144982, -1.192659, -2.680029, -0.839701, 1.570796, 1.715778],accel_mss,speed_ms,0,blend_radius_m)
    movel([0.144651, -1.193163, -2.679793, -0.839433, 1.570796, 1.715448],accel_mss,speed_ms,0,blend_radius_m)
    movel([0.144387, -1.193734, -2.679525, -0.839130, 1.570796, 1.715183],accel_mss,speed_ms,0,blend_radius_m)
    movel([0.144245, -1.194273, -2.679272, -0.838844, 1.570796, 1.715041],accel_mss,speed_ms,0,blend_radius_m)
    movel([0.144134, -1.194666, -2.679087, -0.838635, 1.570796, 1.714931],accel_mss,speed_ms,0,blend_radius_m)
    movel([0.143936, -1.194986, -2.678937, -0.838466, 1.570796, 1.714732],accel_mss,speed_ms,0,blend_radius_m)
    movel([0.143318, -1.195349, -2.678766, -0.838274, 1.570796, 1.714114],accel_mss,speed_ms,0,blend_radius_m)
    speed_ms = 0.003
    movel([0.143132, -1.199044, -2.680560, -0.832785, 1.570796, 1.713928],accel_mss,speed_ms,0,blend_radius_m)
    speed_ms = 0.007
    movel([0.143036, -1.198773, -2.680689, -0.832927, 1.570796, 1.713832],accel_mss,speed_ms,0,blend_radius_m)
    movel([0.143116, -1.198270, -2.680927, -0.833192, 1.570796, 1.713912],accel_mss,speed_ms,0,blend_radius_m)
    movel([0.143455, -1.197078, -2.681489, -0.833822, 1.570796, 1.714251],accel_mss,speed_ms,0,blend_radius_m)
    movel([0.144038, -1.196002, -2.681996, -0.834391, 1.570796, 1.714834],accel_mss,speed_ms,0,blend_radius_m)
    movel([0.144785, -1.195176, -2.682384, -0.834829, 1.570796, 1.715582],accel_mss,speed_ms,0,blend_radius_m)
    movel([0.145608, -1.194685, -2.682614, -0.835090, 1.570796, 1.716404],accel_mss,speed_ms,0,blend_radius_m)
    movel([0.146854, -1.194349, -2.682772, -0.835269, 1.570796, 1.717650],accel_mss,speed_ms,0,blend_radius_m)
    movel([0.148797, -1.194026, -2.682923, -0.835440, 1.570796, 1.719593],accel_mss,speed_ms,0,blend_radius_m)
    movel([0.150703, -1.193786, -2.683035, -0.835568, 1.570796, 1.721499],accel_mss,speed_ms,0,blend_radius_m)
    movel([0.151445, -1.193844, -2.683008, -0.835537, 1.570796, 1.722241],accel_mss,speed_ms,0,blend_radius_m)
    movel([0.151684, -1.194019, -2.682926, -0.835444, 1.570796, 1.722480],accel_mss,speed_ms,0,blend_radius_m)
    movel([0.151798, -1.194309, -2.682790, -0.835290, 1.570796, 1.722594],accel_mss,speed_ms,0,blend_radius_m)
    movel([0.151826, -1.194606, -2.682651, -0.835132, 1.570796, 1.722622],accel_mss,speed_ms,0,blend_radius_m)
    movel([0.151840, -1.195024, -2.682455, -0.834910, 1.570796, 1.722636],accel_mss,speed_ms,0,blend_radius_m)
    movel([0.151696, -1.195570, -2.682199, -0.834620, 1.570796, 1.722492],accel_mss,speed_ms,0,blend_radius_m)
    movel([0.151501, -1.196191, -2.681907, -0.834291, 1.570796, 1.722298],accel_mss,speed_ms,0,blend_radius_m)
    movel([0.151280, -1.196796, -2.681622, -0.833971, 1.570796, 1.722077],accel_mss,speed_ms,0,blend_radius_m)
    movel([0.151065, -1.197294, -2.681388, -0.833708, 1.570796, 1.721862],accel_mss,speed_ms,0,blend_radius_m)
    movel([0.150862, -1.197630, -2.681229, -0.833530, 1.570796, 1.721658],accel_mss,speed_ms,0,blend_radius_m)
    movel([0.150403, -1.197990, -2.681059, -0.833340, 1.570796, 1.721200],accel_mss,speed_ms,0,blend_radius_m)
    movel([0.150113, -1.197993, -2.681057, -0.833338, 1.570796, 1.720910],accel_mss,speed_ms,0,blend_radius_m)
    movel([0.149973, -1.197791, -2.681153, -0.833445, 1.570796, 1.720770],accel_mss,speed_ms,0,blend_radius_m)
    movel([0.150015, -1.197353, -2.681360, -0.833676, 1.570796, 1.720811],accel_mss,speed_ms,0,blend_radius_m)
    movel([0.150240, -1.196681, -2.681676, -0.834031, 1.570796, 1.721036],accel_mss,speed_ms,0,blend_radius_m)
    movel([0.150449, -1.196127, -2.681937, -0.834325, 1.570796, 1.721245],accel_mss,speed_ms,0,blend_radius_m)
    movel([0.150527, -1.195607, -2.682182, -0.834601, 1.570796, 1.721323],accel_mss,speed_ms,0,blend_radius_m)
    movel([0.150292, -1.195152, -2.682395, -0.834842, 1.570796, 1.721089],accel_mss,speed_ms,0,blend_radius_m)
    movel([0.150080, -1.195048, -2.682444, -0.834897, 1.570796, 1.720876],accel_mss,speed_ms,0,blend_radius_m)
    movel([0.149720, -1.195029, -2.682453, -0.834907, 1.570796, 1.720516],accel_mss,speed_ms,0,blend_radius_m)
    movel([0.148947, -1.195091, -2.682424, -0.834874, 1.570796, 1.719743],accel_mss,speed_ms,0,blend_radius_m)
    movel([0.147888, -1.195235, -2.682356, -0.834798, 1.570796, 1.718685],accel_mss,speed_ms,0,blend_radius_m)
    movel([0.146788, -1.195476, -2.682243, -0.834670, 1.570796, 1.717584],accel_mss,speed_ms,0,blend_radius_m)
    movel([0.145823, -1.195752, -2.682113, -0.834523, 1.570796, 1.716619],accel_mss,speed_ms,0,blend_radius_m)
    movel([0.145331, -1.196009, -2.681993, -0.834387, 1.570796, 1.716127],accel_mss,speed_ms,0,blend_radius_m)
    movel([0.144982, -1.196348, -2.681833, -0.834208, 1.570796, 1.715778],accel_mss,speed_ms,0,blend_radius_m)
    movel([0.144651, -1.196851, -2.681596, -0.833942, 1.570796, 1.715448],accel_mss,speed_ms,0,blend_radius_m)
    movel([0.144387, -1.197421, -2.681327, -0.833640, 1.570796, 1.715183],accel_mss,speed_ms,0,blend_radius_m)
    movel([0.144245, -1.197960, -2.681073, -0.833356, 1.570796, 1.715041],accel_mss,speed_ms,0,blend_radius_m)
    movel([0.144134, -1.198353, -2.680888, -0.833149, 1.570796, 1.714931],accel_mss,speed_ms,0,blend_radius_m)
    movel([0.143936, -1.198671, -2.680737, -0.832981, 1.570796, 1.714732],accel_mss,speed_ms,0,blend_radius_m)
    movel([0.143318, -1.199034, -2.680565, -0.832790, 1.570796, 1.714114],accel_mss,speed_ms,0,blend_radius_m)
    speed_ms = 0.003
    movel([0.143132, -1.184515, -2.673317, -0.854557, 1.570796, 1.713928],accel_mss,speed_ms,0,blend_radius_m)
    speed_ms = 1.000
    movel([0.143132, -1.157119, -2.658467, -0.896803, 1.570796, 1.713928],accel_mss,speed_ms,0,blend_radius_m)
    movel([0.116833, -1.199836, -2.638367, -0.874186, 1.570796, 1.687629],accel_mss,speed_ms,0,blend_radius_m)
    movel([0.116833, -1.226889, -2.652654, -0.832845, 1.570796, 1.687629],accel_mss,speed_ms,0,blend_radius_m)
    speed_ms = 0.003
    movel([0.116833, -1.237555, -2.657884, -0.816950, 1.570796, 1.687629],accel_mss,speed_ms,0,blend_radius_m)
    speed_ms = 0.007
    movel([0.117047, -1.237971, -2.657668, -0.816750, 1.570796, 1.687844],accel_mss,speed_ms,0,blend_radius_m)
    movel([0.117087, -1.238384, -2.657453, -0.816551, 1.570796, 1.687884],accel_mss,speed_ms,0,blend_radius_m)
    movel([0.117073, -1.238716, -2.657280, -0.816392, 1.570796, 1.687869],accel_mss,speed_ms,0,blend_radius_m)
    movel([0.116993, -1.239137, -2.657061, -0.816190, 1.570796, 1.687789],accel_mss,speed_ms,0,blend_radius_m)
    movel([0.116788, -1.239942, -2.656642, -0.815805, 1.570796, 1.687584],accel_mss,speed_ms,0,blend_radius_m)
    movel([0.116262, -1.241626, -2.655762, -0.815002, 1.570796, 1.687058],accel_mss,speed_ms,0,blend_radius_m)
    movel([0.115560, -1.243329, -2.654868, -0.814192, 1.570796, 1.686357],accel_mss,speed_ms,0,blend_radius_m)
    movel([0.114825, -1.244785, -2.654101, -0.813503, 1.570796, 1.685621],accel_mss,speed_ms,0,blend_radius_m)
    movel([0.114231, -1.245513, -2.653717, -0.813159, 1.570796, 1.685027],accel_mss,speed_ms,0,blend_radius_m)
    movel([0.112831, -1.246489, -2.653201, -0.812699, 1.570796, 1.683627],accel_mss,speed_ms,0,blend_radius_m)
    movel([0.110772, -1.247488, -2.652671, -0.812230, 1.570796, 1.681568],accel_mss,speed_ms,0,blend_radius_m)
    movel([0.108051, -1.248543, -2.652111, -0.811735, 1.570796, 1.678847],accel_mss,speed_ms,0,blend_radius_m)
    movel([0.104512, -1.249702, -2.651493, -0.811193, 1.570796, 1.675308],accel_mss,speed_ms,0,blend_radius_m)
    movel([0.103009, -1.250155, -2.651251, -0.810982, 1.570796, 1.673805],accel_mss,speed_ms,0,blend_radius_m)
    movel([0.101299, -1.250657, -2.650983, -0.810748, 1.570796, 1.672095],accel_mss,speed_ms,0,blend_radius_m)
    movel([0.099656, -1.251122, -2.650735, -0.810532, 1.570796, 1.670452],accel_mss,speed_ms,0,blend_radius_m)
    movel([0.098359, -1.251475, -2.650546, -0.810368, 1.570796, 1.669156],accel_mss,speed_ms,0,blend_radius_m)
    movel([0.095081, -1.252279, -2.650115, -0.809995, 1.570796, 1.665877],accel_mss,speed_ms,0,blend_radius_m)
    movel([0.093072, -1.252588, -2.649949, -0.809852, 1.570796, 1.663869],accel_mss,speed_ms,0,blend_radius_m)
    movel([0.091832, -1.252507, -2.649993, -0.809889, 1.570796, 1.662629],accel_mss,speed_ms,0,blend_radius_m)
    movel([0.091146, -1.252028, -2.650250, -0.810111, 1.570796, 1.661942],accel_mss,speed_ms,0,blend_radius_m)
    movel([0.090831, -1.250952, -2.650826, -0.810611, 1.570796, 1.661628],accel_mss,speed_ms,0,blend_radius_m)
    movel([0.090806, -1.248846, -2.651950, -0.811594, 1.570796, 1.661602],accel_mss,speed_ms,0,blend_radius_m)
    movel([0.090956, -1.246670, -2.653105, -0.812614, 1.570796, 1.661753],accel_mss,speed_ms,0,blend_radius_m)
    movel([0.091351, -1.245539, -2.653703, -0.813147, 1.570796, 1.662148],accel_mss,speed_ms,0,blend_radius_m)
    movel([0.091708, -1.245070, -2.653951, -0.813368, 1.570796, 1.662504],accel_mss,speed_ms,0,blend_radius_m)
    movel([0.092117, -1.244780, -2.654104, -0.813505, 1.570796, 1.662913],accel_mss,speed_ms,0,blend_radius_m)
    movel([0.092685, -1.244620, -2.654188, -0.813581, 1.570796, 1.663481],accel_mss,speed_ms,0,blend_radius_m)
    movel([0.093614, -1.244549, -2.654226, -0.813614, 1.570796, 1.664411],accel_mss,speed_ms,0,blend_radius_m)
    movel([0.096218, -1.244262, -2.654377, -0.813750, 1.570796, 1.667014],accel_mss,speed_ms,0,blend_radius_m)
    movel([0.099480, -1.243547, -2.654753, -0.814089, 1.570796, 1.670276],accel_mss,speed_ms,0,blend_radius_m)
    movel([0.103447, -1.242410, -2.655350, -0.814628, 1.570796, 1.674243],accel_mss,speed_ms,0,blend_radius_m)
    movel([0.108226, -1.240816, -2.656185, -0.815388, 1.570796, 1.679022],accel_mss,speed_ms,0,blend_radius_m)
    movel([0.110772, -1.239916, -2.656655, -0.815817, 1.570796, 1.681568],accel_mss,speed_ms,0,blend_radius_m)
    movel([0.112222, -1.239378, -2.656936, -0.816075, 1.570796, 1.683018],accel_mss,speed_ms,0,blend_radius_m)
    movel([0.113204, -1.238973, -2.657147, -0.816269, 1.570796, 1.684000],accel_mss,speed_ms,0,blend_radius_m)
    movel([0.114008, -1.238576, -2.657354, -0.816460, 1.570796, 1.684804],accel_mss,speed_ms,0,blend_radius_m)
    movel([0.115583, -1.237757, -2.657779, -0.816853, 1.570796, 1.686380],accel_mss,speed_ms,0,blend_radius_m)
    movel([0.116394, -1.237472, -2.657927, -0.816990, 1.570796, 1.687190],accel_mss,speed_ms,0,blend_radius_m)
    movel([0.116833, -1.237555, -2.657884, -0.816950, 1.570796, 1.687629],accel_mss,speed_ms,0,blend_radius_m)
    speed_ms = 0.003
    movel([0.116833, -1.241175, -2.659611, -0.811603, 1.570796, 1.687629],accel_mss,speed_ms,0,blend_radius_m)
    speed_ms = 0.007
    movel([0.117047, -1.241590, -2.659394, -0.811405, 1.570796, 1.687844],accel_mss,speed_ms,0,blend_radius_m)
    movel([0.117087, -1.242003, -2.659179, -0.811207, 1.570796, 1.687884],accel_mss,speed_ms,0,blend_radius_m)
    movel([0.117073, -1.242334, -2.659005, -0.811049, 1.570796, 1.687869],accel_mss,speed_ms,0,blend_radius_m)
    movel([0.116993, -1.242754, -2.658786, -0.810849, 1.570796, 1.687789],accel_mss,speed_ms,0,blend_radius_m)
    movel([0.116788, -1.243558, -2.658365, -0.810466, 1.570796, 1.687584],accel_mss,speed_ms,0,blend_radius_m)
    movel([0.116262, -1.245238, -2.657482, -0.809669, 1.570796, 1.687058],accel_mss,speed_ms,0,blend_radius_m)
    movel([0.115560, -1.246939, -2.656585, -0.808865, 1.570796, 1.686357],accel_mss,speed_ms,0,blend_radius_m)
    movel([0.114825, -1.248392, -2.655816, -0.808181, 1.570796, 1.685621],accel_mss,speed_ms,0,blend_radius_m)
    movel([0.114231, -1.249119, -2.655430, -0.807840, 1.570796, 1.685027],accel_mss,speed_ms,0,blend_radius_m)
    movel([0.112831, -1.250093, -2.654912, -0.807384, 1.570796, 1.683627],accel_mss,speed_ms,0,blend_radius_m)
    movel([0.110772, -1.251090, -2.654381, -0.806918, 1.570796, 1.681568],accel_mss,speed_ms,0,blend_radius_m)
    movel([0.108051, -1.252143, -2.653819, -0.806427, 1.570796, 1.678847],accel_mss,speed_ms,0,blend_radius_m)
    movel([0.104512, -1.253300, -2.653199, -0.805889, 1.570796, 1.675308],accel_mss,speed_ms,0,blend_radius_m)
    movel([0.103009, -1.253752, -2.652957, -0.805680, 1.570796, 1.673805],accel_mss,speed_ms,0,blend_radius_m)
    movel([0.101299, -1.254253, -2.652688, -0.805448, 1.570796, 1.672095],accel_mss,speed_ms,0,blend_radius_m)
    movel([0.099656, -1.254718, -2.652438, -0.805233, 1.570796, 1.670452],accel_mss,speed_ms,0,blend_radius_m)
    movel([0.098359, -1.255070, -2.652249, -0.805070, 1.570796, 1.669156],accel_mss,speed_ms,0,blend_radius_m)
    movel([0.095081, -1.255872, -2.651817, -0.804700, 1.570796, 1.665877],accel_mss,speed_ms,0,blend_radius_m)
    movel([0.093072, -1.256180, -2.651651, -0.804558, 1.570796, 1.663869],accel_mss,speed_ms,0,blend_radius_m)
    movel([0.091832, -1.256100, -2.651694, -0.804595, 1.570796, 1.662629],accel_mss,speed_ms,0,blend_radius_m)
    movel([0.091146, -1.255621, -2.651952, -0.804816, 1.570796, 1.661942],accel_mss,speed_ms,0,blend_radius_m)
    movel([0.090831, -1.254548, -2.652530, -0.805311, 1.570796, 1.661628],accel_mss,speed_ms,0,blend_radius_m)
    movel([0.090806, -1.252445, -2.653657, -0.806286, 1.570796, 1.661602],accel_mss,speed_ms,0,blend_radius_m)
    movel([0.090956, -1.250273, -2.654817, -0.807299, 1.570796, 1.661753],accel_mss,speed_ms,0,blend_radius_m)
    movel([0.091351, -1.249145, -2.655416, -0.807828, 1.570796, 1.662148],accel_mss,speed_ms,0,blend_radius_m)
    movel([0.091708, -1.248676, -2.655665, -0.808048, 1.570796, 1.662504],accel_mss,speed_ms,0,blend_radius_m)
    movel([0.092117, -1.248386, -2.655819, -0.808184, 1.570796, 1.662913],accel_mss,speed_ms,0,blend_radius_m)
    movel([0.092685, -1.248227, -2.655903, -0.808259, 1.570796, 1.663481],accel_mss,speed_ms,0,blend_radius_m)
    movel([0.093614, -1.248156, -2.655941, -0.808292, 1.570796, 1.664411],accel_mss,speed_ms,0,blend_radius_m)
    movel([0.096218, -1.247870, -2.656093, -0.808427, 1.570796, 1.667014],accel_mss,speed_ms,0,blend_radius_m)
    movel([0.099480, -1.247156, -2.656470, -0.808763, 1.570796, 1.670276],accel_mss,speed_ms,0,blend_radius_m)
    movel([0.103447, -1.246022, -2.657069, -0.809298, 1.570796, 1.674243],accel_mss,speed_ms,0,blend_radius_m)
    movel([0.108226, -1.244430, -2.657907, -0.810052, 1.570796, 1.679022],accel_mss,speed_ms,0,blend_radius_m)
    movel([0.110772, -1.243532, -2.658378, -0.810479, 1.570796, 1.681568],accel_mss,speed_ms,0,blend_radius_m)
    movel([0.112222, -1.242995, -2.658660, -0.810735, 1.570796, 1.683018],accel_mss,speed_ms,0,blend_radius_m)
    movel([0.113204, -1.242590, -2.658872, -0.810927, 1.570796, 1.684000],accel_mss,speed_ms,0,blend_radius_m)
    movel([0.114008, -1.242194, -2.659079, -0.811116, 1.570796, 1.684804],accel_mss,speed_ms,0,blend_radius_m)
    movel([0.115583, -1.241377, -2.659505, -0.811507, 1.570796, 1.686380],accel_mss,speed_ms,0,blend_radius_m)
    movel([0.116394, -1.241092, -2.659654, -0.811643, 1.570796, 1.687190],accel_mss,speed_ms,0,blend_radius_m)
    movel([0.116833, -1.241175, -2.659611, -0.811603, 1.570796, 1.687629],accel_mss,speed_ms,0,blend_radius_m)
    speed_ms = 0.003
    movel([0.116833, -1.226889, -2.652654, -0.832845, 1.570796, 1.687629],accel_mss,speed_ms,0,blend_radius_m)
    speed_ms = 1.000
    movel([0.116833, -1.199836, -2.638367, -0.874186, 1.570796, 1.687629],accel_mss,speed_ms,0,blend_radius_m)
    movel([0.120445, -1.198045, -2.639248, -0.875095, 1.570796, 1.691242],accel_mss,speed_ms,0,blend_radius_m)
    movel([0.120445, -1.225115, -2.653559, -0.833714, 1.570796, 1.691242],accel_mss,speed_ms,0,blend_radius_m)
    speed_ms = 0.003
    movel([0.120445, -1.235790, -2.658798, -0.817801, 1.570796, 1.691242],accel_mss,speed_ms,0,blend_radius_m)
    speed_ms = 0.007
    movel([0.119507, -1.238641, -2.657320, -0.816429, 1.570796, 1.690304],accel_mss,speed_ms,0,blend_radius_m)
    movel([0.118536, -1.241261, -2.655953, -0.815176, 1.570796, 1.689333],accel_mss,speed_ms,0,blend_radius_m)
    movel([0.117534, -1.243652, -2.654698, -0.814039, 1.570796, 1.688331],accel_mss,speed_ms,0,blend_radius_m)
    movel([0.117009, -1.244810, -2.654088, -0.813491, 1.570796, 1.687805],accel_mss,speed_ms,0,blend_radius_m)
    movel([0.116695, -1.245417, -2.653768, -0.813204, 1.570796, 1.687491],accel_mss,speed_ms,0,blend_radius_m)
    movel([0.116436, -1.245798, -2.653567, -0.813025, 1.570796, 1.687232],accel_mss,speed_ms,0,blend_radius_m)
    movel([0.116154, -1.246077, -2.653419, -0.812893, 1.570796, 1.686950],accel_mss,speed_ms,0,blend_radius_m)
    movel([0.114416, -1.247109, -2.652872, -0.812408, 1.570796, 1.685212],accel_mss,speed_ms,0,blend_radius_m)
    movel([0.110469, -1.248706, -2.652024, -0.811659, 1.570796, 1.681265],accel_mss,speed_ms,0,blend_radius_m)
    movel([0.105892, -1.250368, -2.651138, -0.810883, 1.570796, 1.676688],accel_mss,speed_ms,0,blend_radius_m)
    movel([0.101275, -1.251838, -2.650351, -0.810199, 1.570796, 1.672071],accel_mss,speed_ms,0,blend_radius_m)
    movel([0.097010, -1.253016, -2.649720, -0.809654, 1.570796, 1.667806],accel_mss,speed_ms,0,blend_radius_m)
    movel([0.093314, -1.253841, -2.649276, -0.809272, 1.570796, 1.664111],accel_mss,speed_ms,0,blend_radius_m)
    movel([0.090388, -1.254324, -2.649016, -0.809049, 1.570796, 1.661185],accel_mss,speed_ms,0,blend_radius_m)
    movel([0.089540, -1.254068, -2.649153, -0.809167, 1.570796, 1.660336],accel_mss,speed_ms,0,blend_radius_m)
    movel([0.088883, -1.252023, -2.650252, -0.810114, 1.570796, 1.659679],accel_mss,speed_ms,0,blend_radius_m)
    movel([0.089050, -1.244273, -2.654371, -0.813745, 1.570796, 1.659846],accel_mss,speed_ms,0,blend_radius_m)
    movel([0.089536, -1.236364, -2.658501, -0.817524, 1.570796, 1.660332],accel_mss,speed_ms,0,blend_radius_m)
    movel([0.090414, -1.230909, -2.661307, -0.820173, 1.570796, 1.661211],accel_mss,speed_ms,0,blend_radius_m)
    movel([0.090708, -1.229904, -2.661820, -0.820665, 1.570796, 1.661505],accel_mss,speed_ms,0,blend_radius_m)
    movel([0.091054, -1.229331, -2.662112, -0.820946, 1.570796, 1.661850],accel_mss,speed_ms,0,blend_radius_m)
    movel([0.091650, -1.228821, -2.662372, -0.821197, 1.570796, 1.662446],accel_mss,speed_ms,0,blend_radius_m)
    movel([0.093003, -1.227990, -2.662794, -0.821605, 1.570796, 1.663799],accel_mss,speed_ms,0,blend_radius_m)
    movel([0.095187, -1.226778, -2.663409, -0.822202, 1.570796, 1.665983],accel_mss,speed_ms,0,blend_radius_m)
    movel([0.097230, -1.225790, -2.663908, -0.822691, 1.570796, 1.668026],accel_mss,speed_ms,0,blend_radius_m)
    movel([0.099701, -1.224762, -2.664427, -0.823200, 1.570796, 1.670497],accel_mss,speed_ms,0,blend_radius_m)
    movel([0.103416, -1.223367, -2.665129, -0.823893, 1.570796, 1.674212],accel_mss,speed_ms,0,blend_radius_m)
    movel([0.108750, -1.221528, -2.666052, -0.824810, 1.570796, 1.679546],accel_mss,speed_ms,0,blend_radius_m)
    movel([0.113497, -1.220122, -2.666754, -0.825513, 1.570796, 1.684294],accel_mss,speed_ms,0,blend_radius_m)
    movel([0.117730, -1.219129, -2.667249, -0.826011, 1.570796, 1.688526],accel_mss,speed_ms,0,blend_radius_m)
    movel([0.121518, -1.218530, -2.667547, -0.826313, 1.570796, 1.692314],accel_mss,speed_ms,0,blend_radius_m)
    movel([0.122546, -1.218462, -2.667580, -0.826347, 1.570796, 1.693342],accel_mss,speed_ms,0,blend_radius_m)
    movel([0.122998, -1.218611, -2.667506, -0.826272, 1.570796, 1.693794],accel_mss,speed_ms,0,blend_radius_m)
    movel([0.123197, -1.219033, -2.667296, -0.826059, 1.570796, 1.693993],accel_mss,speed_ms,0,blend_radius_m)
    movel([0.123242, -1.220065, -2.666782, -0.825541, 1.570796, 1.694038],accel_mss,speed_ms,0,blend_radius_m)
    movel([0.123245, -1.220596, -2.666518, -0.825276, 1.570796, 1.694042],accel_mss,speed_ms,0,blend_radius_m)
    movel([0.123250, -1.221075, -2.666278, -0.825036, 1.570796, 1.694046],accel_mss,speed_ms,0,blend_radius_m)
    movel([0.123256, -1.221474, -2.666079, -0.824837, 1.570796, 1.694052],accel_mss,speed_ms,0,blend_radius_m)
    movel([0.123267, -1.221758, -2.665937, -0.824695, 1.570796, 1.694063],accel_mss,speed_ms,0,blend_radius_m)
    movel([0.123104, -1.222963, -2.665332, -0.824094, 1.570796, 1.693901],accel_mss,speed_ms,0,blend_radius_m)
    movel([0.122915, -1.224347, -2.664636, -0.823406, 1.570796, 1.693712],accel_mss,speed_ms,0,blend_radius_m)
    movel([0.122686, -1.225949, -2.663828, -0.822612, 1.570796, 1.693482],accel_mss,speed_ms,0,blend_radius_m)
